# B&R Automation Studio project Praktyki_12_08
Automation Studio 4.12.5.95 SP; technology packages: mappCockpit 5.24.3, mappMotion 5.26.1, mappView 5.24.2

## Configuration Config1

CPU X20CP0484-1, AutomationRuntime K4.93, Build 4.1.2, Safety 0.0, Vc V4.72.6

### Task classes (Cpu.sw)
```
Cyclic#1:
  TCPXYZ <- PickAndPlace.TCPXYZ.prg
  Program <- PickAndPlace.Program.prg [disabled]
  PrgMechs <- PickAndPlace.PrgMechs.prg [disabled]
  PrgPickCor <- PickAndPlace.PrgPickCore.prg
  PrgPick <- PickAndPlace.PrgPick.prg
  PrgPlace <- PickAndPlace.PrgPlace.prg
DataObjects: McAcpSys
NcDataObjects: McDriveLog
Binaries: udbdef, arsvcreg, FWRules, McAcpDrv, McMechSys, McAcpSim, TCData, arflatprv, arcoal, visionUnit, mvLoader, McProfGen, mCoWebSc, TCLang, iomap, Config_4, asfw, Config_9, Config_3, Role, Config_8, Config_6, Config_7, Config_5, Config_1, Config_2, arconfig, ashwac, ashwd, Hierarchy, sysconf, User, Settings, Config_11, Config_10, Settings_1, viApp, viComp, Config_12, Config_13, Config
Libraries: McBase, MpBase, MpRobotics, McAxGroup, McPathGen, McAxis, McProgInt, McAcpAx, MpAxis, UserLib, MpPick, McTrkPath, CoTrace, AsZip, FileIO, runtime, Library, ViBase, AsARCfg, powerlnk, AsEPL, AsIO, sys_lib, DataObj, astime, McPureVAx, MpAlarmX, asmem, brsystem, asarprof, asarlog, asieccon, arssl
```

### Task classes (Cpu.sw)
```
Cyclic#4:
  PrgMechs <- PickAndPlace.PrgMechs.prg
  PrgPick <- PickAndPlace.PrgPick.prg
  PrgPlace <- PickAndPlace.PrgPlace.prg
  PrgPickCor <- PickAndPlace.PrgPickCore.prg
DataObjects: McAcpSys
NcDataObjects: McDriveLog
Binaries: McAcpDrv, udbdef, McAcpSim, mvLoader, arflatprv, McMechSys, TCData, mCoWebSc, FWRules, arcoal, arsvcreg, Settings, iomap, TraceConfi, ashwac, asfw, sysconf, arconfig, Config_6, Config_8, Hierarchy, ashwd, Role, Config_7, User, Config_9, Config_3, Config_1, Config_4, Config_2, Config_5, Config_14, Config_12, Config_10, Config_13, Config_11
Libraries: McBase, MpBase, MpRobotics, McAxGroup, McPathGen, McAxis, McProgInt, McAcpAx, CoTrace, AsZip, FileIO, runtime, MpAxis, MpPick, McTrkPath, asarprof, asieccon, asarlog, asio, asmem, astime, dataobj, asepl, brsystem, arssl, sys_lib, powerlnk
```

### Hardware
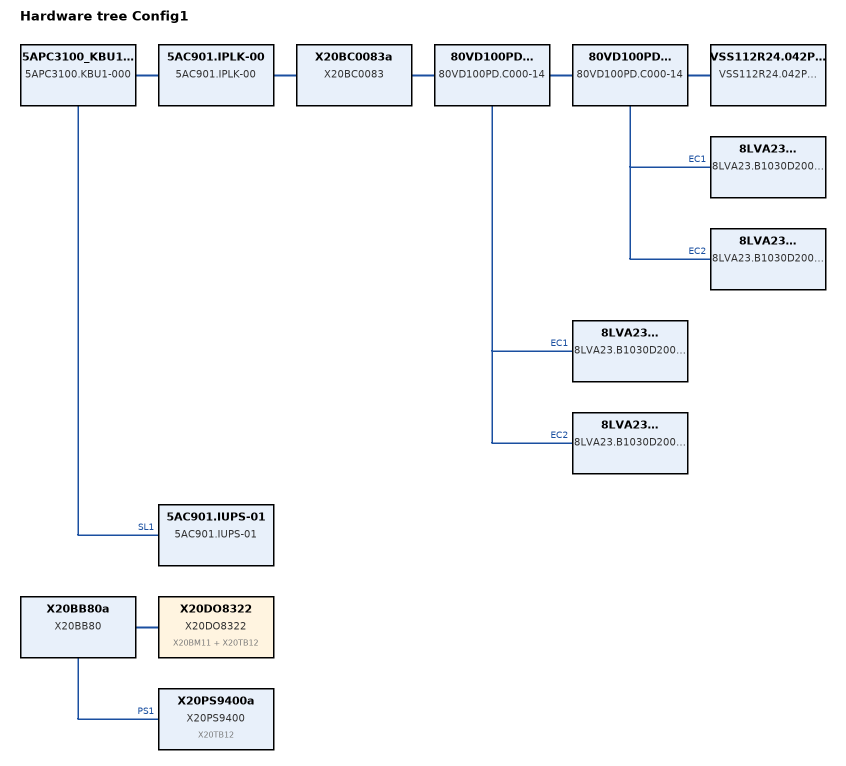
```
5AC901.IPLK-00 : 5AC901.IPLK-00 v1.8.0.1  [SL -> 5APC3100_KBU1_000.SL2]
  Connector IF1:
    MtuSize = 1500
    Channel1
    ChannelID1 = McAcpBroadcast
    ChannelType1 = OCTET[96]
    InternetAddress = 12.10.10.240
    SubnetMask = 255.255.255.0
5AC901.IUPS-01 : 5AC901.IUPS-01 v1.3.1.0  [SL -> 5APC3100_KBU1_000.SL1]
5APC3100_KBU1_000 : 5APC3100.KBU1-000 v2.2.1.0
  Connector IF3:
    AssignedOperatingSystem = ARemb
    ActivateDevice = 1
    Mode = Manual
    InternetAddress = 10.0.0.150
    SubnetMask = 255.255.255.0
    ActivateSnmp = 2
  Connector IF4:
    AssignedOperatingSystem = ARemb
    ActivateDevice = 1
    Mode = Manual
    InternetAddress = 192.168.0.20
    SubnetMask = 255.255.255.0
    ActivateSnmp = 2
  Connector IF5:
    AssignedOperatingSystem = ARemb
  Connector IF6:
    AssignedOperatingSystem = ARemb
  Connector IF7:
    AssignedOperatingSystem = ARemb
  Connector IF8:
    AssignedOperatingSystem = ARemb
  ConfigurationID = prawdziwaDelta_Config1
  Simulation = 1
  TimerDeviceType = EPLX2X
  TimerDevice = 5AC901.IPLK-00.IF1
  TaskClassIdleTime = 2000
  Cyclic1Tolerance = 0
  FileDevice1
  FileDeviceName1 = CNC_PrgDir
  FileDevicePath1 = USER_PATH
  FtpUser1
  FtpUsername1 = admin
  FtpUserPassword1 = q3LIg5ZPX9qKnYfEoKnLCuwwHRw0InMkB5MY3lkoy6s=
  FtpUserSalt1 = imXNidk5
  FTPAccessRight1 = 0
  ActivateOpcUa = 1
  OpcUaInformationModels_PV_Version = 1
80VD100PD.C000-14 : 80VD100PD.C000-14 v2.5.0.0  [PLK1 -> X20BC0083a.PLK2 (NodeNumber=1) [Cable Type=PowerlinkCable, Length=10, Version=1.0.0.3]; PLK2 -> 80VD100PD.C000-14a.PLK1 (NodeNumber=1) [Cable Type=PowerlinkCable, Length=10, Version=1.0.0.3]; EC1 -> 8LVA23.B1030D200-0.EC; EC2 -> 8LVA23.B1030D200-0a.EC; MT2 -> 8LVA23.B1030D200-0a.MT]
  DriveConfiguration/Module:
    McAcoposTypeID = AcoposMicroDConfig
    ActivateACOPOSSimulationOnPLC = 0
  DriveConfiguration/Channel[1]/RealAxis:
    AxisReference = gAxisQ1
    MechanicalElementsIsInvisible = 0
  DriveConfiguration/Channel[1]/RealAxis/MechanicalElements/Gearbox:
    InputIsReadOnly = 0
    Input = 25
    OutputIsReadOnly = 0
    Output = 1
  DriveConfiguration/Channel[1]/RealAxis/MechanicalElements/RotaryToLinearTransformation:
    ReferenceDistanceIsReadOnly = 0
    ReferenceDistance = 1
  DriveConfiguration/Channel[1]/RealAxis/Controller:
    ModeIsReadOnly = 0
    Mode = PositionController
  DriveConfiguration/Channel[1]/RealAxis/Controller/Mode/Position:
    ProportionalGain = 402
    IntegrationTime = 0.0
    PredictionTime = 0.0004
    TotalDelayTime = 0.0004
  DriveConfiguration/Channel[1]/RealAxis/Controller/Mode/Speed:
    ProportionalGainIsReadOnly = 0
    ProportionalGain = 1.7
    IntegrationTimeIsReadOnly = 0
    IntegrationTime = 0.0
    FilterTimeIsReadOnly = 0
    FilterTime = 0.0
  DriveConfiguration/Channel[1]/RealAxis/Controller/Mode/LoopFilters:
    LoopFilterXIsReadOnly = 0
    LoopFilter1 = NotUsed
    LoopFilter2 = NotUsed
    LoopFilter3 = NotUsed
  DriveConfiguration/Channel[1]/RealAxis/Homing:
    ModeIsReadOnly = 0
    Mode = Absolute
  DriveConfiguration/Channel[1]/RealAxis/Homing/Mode:
    Position = 0
  DriveConfiguration/Channel[1]/RealAxis/Homing:
    RestorePositionVariable = 
  DriveConfiguration/Channel[1]/RealAxis/StopReaction:
    QuickstopIsReadOnly = 0
    Quickstop = DecelerationLimit
    DriveErrorIsReadOnly = 0
    DriveError = DecelerationLimit
  DriveConfiguration/Channel[1]/RealAxis/MovementErrorLimits:
    PositionError = 1.0
    VelocityErrorMonitoring = Automatic1
  DriveConfiguration/Channel[1]/RealAxis:
    JerkFilterIsReadOnly = 0
    JerkFilter = NotUsed
    ZeroVibrationFilter = NotUsed
  DriveConfiguration/Channel[1]/RealAxis/DigitalInputs/HomingSwitch:
    SourceIsReadOnly = 0
    Source = NotUsed
    Level = High
  DriveConfiguration/Channel[1]/RealAxis/DigitalInputs/PositiveLimitSwitch:
    SourceIsReadOnly = 0
    Source = NotUsed
    Level = High
  DriveConfiguration/Channel[1]/RealAxis/DigitalInputs/NegativeLimitSwitch:
    SourceIsReadOnly = 0
    Source = NotUsed
    Level = High
  DriveConfiguration/Channel[1]/RealAxis/DigitalInputs/Trigger1:
    Source = X2Trigger1
    Level = High
  DriveConfiguration/Channel[1]/RealAxis/DigitalInputs/Trigger2:
    Source = X2Trigger2
    Level = High
  DriveConfiguration/Channel[1]/RealAxis/DigitalInputs/Quickstop:
    Input = Trigger2
  DriveConfiguration/Channel[1]/RealAxis/Simulation:
    SimulationModeOnPLC = SetValueGeneration
    SimulationModeOnACOPOS = NotUsed
  DriveConfiguration/Channel[1]:
    ExternalEncoderAxis = NotUsed
  DriveConfiguration/Channel[2]/RealAxis:
    AxisReference = gAxisQ2
    MechanicalElementsIsInvisible = 0
  DriveConfiguration/Channel[2]/RealAxis/MechanicalElements/Gearbox:
    InputIsReadOnly = 0
    Input = 25
    OutputIsReadOnly = 0
    Output = 1
  DriveConfiguration/Channel[2]/RealAxis/MechanicalElements/RotaryToLinearTransformation:
    ReferenceDistanceIsReadOnly = 0
    ReferenceDistance = 1
  DriveConfiguration/Channel[2]/RealAxis/Controller:
    ModeIsReadOnly = 0
    Mode = PositionController
  DriveConfiguration/Channel[2]/RealAxis/Controller/Mode/Position:
    ProportionalGain = 393
    IntegrationTime = 0.0
    PredictionTime = 0.0004
    TotalDelayTime = 0.0004
  DriveConfiguration/Channel[2]/RealAxis/Controller/Mode/Speed:
    ProportionalGainIsReadOnly = 0
    ProportionalGain = 1.65
    IntegrationTimeIsReadOnly = 0
    IntegrationTime = 0.0
    FilterTimeIsReadOnly = 0
    FilterTime = 0.0
  DriveConfiguration/Channel[2]/RealAxis/Controller/Mode/LoopFilters:
    LoopFilterXIsReadOnly = 0
    LoopFilter1 = NotUsed
    LoopFilter2 = NotUsed
    LoopFilter3 = NotUsed
  DriveConfiguration/Channel[2]/RealAxis/Homing:
    ModeIsReadOnly = 0
    Mode = Absolute
  DriveConfiguration/Channel[2]/RealAxis/Homing/Mode:
    Position = 0
  DriveConfiguration/Channel[2]/RealAxis/Homing:
    RestorePositionVariable = 
  DriveConfiguration/Channel[2]/RealAxis/StopReaction:
    QuickstopIsReadOnly = 0
    Quickstop = DecelerationLimit
    DriveErrorIsReadOnly = 0
    DriveError = DecelerationLimit
  DriveConfiguration/Channel[2]/RealAxis/MovementErrorLimits:
    PositionError = 1.0
    VelocityErrorMonitoring = Automatic1
  DriveConfiguration/Channel[2]/RealAxis:
    JerkFilterIsReadOnly = 0
    JerkFilter = NotUsed
    ZeroVibrationFilter = NotUsed
  DriveConfiguration/Channel[2]/RealAxis/DigitalInputs/HomingSwitch:
    SourceIsReadOnly = 0
    Source = NotUsed
    Level = High
  DriveConfiguration/Channel[2]/RealAxis/DigitalInputs/PositiveLimitSwitch:
    SourceIsReadOnly = 0
    Source = NotUsed
    Level = High
  DriveConfiguration/Channel[2]/RealAxis/DigitalInputs/NegativeLimitSwitch:
    SourceIsReadOnly = 0
    Source = NotUsed
    Level = High
  DriveConfiguration/Channel[2]/RealAxis/DigitalInputs/Trigger1:
    Source = X2Trigger1
    Level = High
  DriveConfiguration/Channel[2]/RealAxis/DigitalInputs/Trigger2:
    Source = X2Trigger2
    Level = High
  DriveConfiguration/Channel[2]/RealAxis/DigitalInputs/Quickstop:
    Input = Trigger2
  DriveConfiguration/Channel[2]/RealAxis/Simulation:
    SimulationModeOnPLC = SetValueGeneration
    SimulationModeOnACOPOS = NotUsed
  DriveConfiguration/Channel[2]:
    ExternalEncoderAxis = NotUsed
80VD100PD.C000-14a : 80VD100PD.C000-14 v2.5.0.0  [PLK1 -> 80VD100PD.C000-14.PLK2 (NodeNumber=2) [Cable Type=PowerlinkCable, Length=10, Version=1.0.0.3]; PLK2 -> VSS112R24.042P-000.PLK1 (NodeNumber=2) [Cable Type=PowerlinkCable, Length=10, Version=1.0.0.3]; EC1 -> 8LVA23.B1030D200-0b.EC; EC2 -> 8LVA23.B1030D200-0c.EC; MT2 -> 8LVA23.B1030D200-0c.MT]
  DriveConfiguration/Module:
    McAcoposTypeID = AcoposMicroDConfig
    ActivateACOPOSSimulationOnPLC = 0
  DriveConfiguration/Channel[1]/RealAxis:
    AxisReference = gAxisQ3
    MechanicalElementsIsInvisible = 0
  DriveConfiguration/Channel[1]/RealAxis/MechanicalElements/Gearbox:
    InputIsReadOnly = 0
    Input = 25
    OutputIsReadOnly = 0
    Output = 1
  DriveConfiguration/Channel[1]/RealAxis/MechanicalElements/RotaryToLinearTransformation:
    ReferenceDistanceIsReadOnly = 0
    ReferenceDistance = 1
  DriveConfiguration/Channel[1]/RealAxis/Controller:
    ModeIsReadOnly = 0
    Mode = PositionController
  DriveConfiguration/Channel[1]/RealAxis/Controller/Mode/Position:
    ProportionalGain = 400
    IntegrationTime = 0.0
    PredictionTime = 0.0004
    TotalDelayTime = 0.0004
  DriveConfiguration/Channel[1]/RealAxis/Controller/Mode/Speed:
    ProportionalGainIsReadOnly = 0
    ProportionalGain = 1.7
    IntegrationTimeIsReadOnly = 0
    IntegrationTime = 0.0
    FilterTimeIsReadOnly = 0
    FilterTime = 0.0
  DriveConfiguration/Channel[1]/RealAxis/Controller/Mode/LoopFilters:
    LoopFilterXIsReadOnly = 0
    LoopFilter1 = NotUsed
    LoopFilter2 = NotUsed
    LoopFilter3 = NotUsed
  DriveConfiguration/Channel[1]/RealAxis/Homing:
    ModeIsReadOnly = 0
    Mode = Absolute
  DriveConfiguration/Channel[1]/RealAxis/Homing/Mode:
    Position = 0
  DriveConfiguration/Channel[1]/RealAxis/Homing:
    RestorePositionVariable = 
  DriveConfiguration/Channel[1]/RealAxis/StopReaction:
    QuickstopIsReadOnly = 0
    Quickstop = DecelerationLimit
    DriveErrorIsReadOnly = 0
    DriveError = DecelerationLimit
  DriveConfiguration/Channel[1]/RealAxis/MovementErrorLimits:
    PositionError = 1.0
    VelocityErrorMonitoring = Automatic1
  DriveConfiguration/Channel[1]/RealAxis:
    JerkFilterIsReadOnly = 0
    JerkFilter = NotUsed
    ZeroVibrationFilter = NotUsed
  DriveConfiguration/Channel[1]/RealAxis/DigitalInputs/HomingSwitch:
    SourceIsReadOnly = 0
    Source = NotUsed
    Level = High
  DriveConfiguration/Channel[1]/RealAxis/DigitalInputs/PositiveLimitSwitch:
    SourceIsReadOnly = 0
    Source = NotUsed
    Level = High
  DriveConfiguration/Channel[1]/RealAxis/DigitalInputs/NegativeLimitSwitch:
    SourceIsReadOnly = 0
    Source = NotUsed
    Level = High
  DriveConfiguration/Channel[1]/RealAxis/DigitalInputs/Trigger1:
    Source = X2Trigger1
    Level = High
  DriveConfiguration/Channel[1]/RealAxis/DigitalInputs/Trigger2:
    Source = X2Trigger2
    Level = High
  DriveConfiguration/Channel[1]/RealAxis/DigitalInputs/Quickstop:
    Input = Trigger2
  DriveConfiguration/Channel[1]/RealAxis/Simulation:
    SimulationModeOnPLC = SetValueGeneration
    SimulationModeOnACOPOS = NotUsed
  DriveConfiguration/Channel[1]:
    ExternalEncoderAxis = NotUsed
  DriveConfiguration/Channel[2]/RealAxis:
    AxisReference = gAxis_1
    MechanicalElementsIsInvisible = 0
  DriveConfiguration/Channel[2]/RealAxis/MechanicalElements/Gearbox:
    InputIsReadOnly = 0
    Input = 1
    OutputIsReadOnly = 0
    Output = 1
  DriveConfiguration/Channel[2]/RealAxis/MechanicalElements/RotaryToLinearTransformation:
    ReferenceDistanceIsReadOnly = 0
    ReferenceDistance = 1
  DriveConfiguration/Channel[2]/RealAxis/Controller:
    ModeIsReadOnly = 0
    Mode = PositionController
  DriveConfiguration/Channel[2]/RealAxis/Controller/Mode/Position:
    ProportionalGain = 50.0
    IntegrationTime = 0.0
    PredictionTime = 0.0004
    TotalDelayTime = 0.0004
  DriveConfiguration/Channel[2]/RealAxis/Controller/Mode/Speed:
    ProportionalGainIsReadOnly = 0
    ProportionalGain = 2.0
    IntegrationTimeIsReadOnly = 0
    IntegrationTime = 0.0
    FilterTimeIsReadOnly = 0
    FilterTime = 0.0
  DriveConfiguration/Channel[2]/RealAxis/Controller/Mode/LoopFilters:
    LoopFilterXIsReadOnly = 0
    LoopFilter1 = NotUsed
    LoopFilter2 = NotUsed
    LoopFilter3 = NotUsed
  DriveConfiguration/Channel[2]/RealAxis/Homing:
    ModeIsReadOnly = 0
    Mode = Direct
  DriveConfiguration/Channel[2]/RealAxis/Homing/Mode:
    Position = 0.0
    ReferencePulse = NotUsed
  DriveConfiguration/Channel[2]/RealAxis/Homing:
    RestorePositionVariable = 
  DriveConfiguration/Channel[2]/RealAxis/StopReaction:
    QuickstopIsReadOnly = 0
    Quickstop = DecelerationLimit
    DriveErrorIsReadOnly = 0
    DriveError = DecelerationLimit
  DriveConfiguration/Channel[2]/RealAxis/MovementErrorLimits:
    PositionError = 1.0
    VelocityErrorMonitoring = Automatic1
  DriveConfiguration/Channel[2]/RealAxis:
    JerkFilterIsReadOnly = 0
    JerkFilter = NotUsed
    ZeroVibrationFilter = NotUsed
  DriveConfiguration/Channel[2]/RealAxis/DigitalInputs/HomingSwitch:
    SourceIsReadOnly = 0
    Source = NotUsed
    Level = High
  DriveConfiguration/Channel[2]/RealAxis/DigitalInputs/PositiveLimitSwitch:
    SourceIsReadOnly = 0
    Source = NotUsed
    Level = High
  DriveConfiguration/Channel[2]/RealAxis/DigitalInputs/NegativeLimitSwitch:
    SourceIsReadOnly = 0
    Source = NotUsed
    Level = High
  DriveConfiguration/Channel[2]/RealAxis/DigitalInputs/Trigger1:
    Source = X2Trigger1
    Level = High
  DriveConfiguration/Channel[2]/RealAxis/DigitalInputs/Trigger2:
    Source = X2Trigger2
    Level = High
  DriveConfiguration/Channel[2]/RealAxis/DigitalInputs/Quickstop:
    Input = Trigger2
  DriveConfiguration/Channel[2]/RealAxis/Simulation:
    SimulationModeOnPLC = SetValueGeneration
    SimulationModeOnACOPOS = NotUsed
  DriveConfiguration/Channel[2]:
    ExternalEncoderAxis = NotUsed
8LVA23.B1030D200-0 : 8LVA23.B1030D200-0 v2.2.0.3  [EC -> 80VD100PD.C000-14.EC1; MT -> 80VD100PD.C000-14.MT1]
  M1/MotorParameters:
    MOTOR_AMB_TEMP_RATED = 40
8LVA23.B1030D200-0a : 8LVA23.B1030D200-0 v2.2.0.3  [EC -> 80VD100PD.C000-14.EC2; MT -> 80VD100PD.C000-14.MT2]
  M1/MotorParameters:
    MOTOR_AMB_TEMP_RATED = 40
8LVA23.B1030D200-0b : 8LVA23.B1030D200-0 v2.2.0.3  [EC -> 80VD100PD.C000-14a.EC1; MT -> 80VD100PD.C000-14a.MT1]
  M1/MotorParameters:
    MOTOR_AMB_TEMP_RATED = 40
8LVA23.B1030D200-0c : 8LVA23.B1030D200-0 v2.2.0.3  [EC -> 80VD100PD.C000-14a.EC2; MT -> 80VD100PD.C000-14a.MT2]
  M1/MotorParameters:
    MOTOR_AMB_TEMP_RATED = 40
VSS112R24.042P-000 : VSS112R24.042P-000 v1.9.0.730  [PLK1 -> 80VD100PD.C000-14a.PLK2 (NodeNumber=4) [Cable Type=PowerlinkCable, Length=10, Version=1.0.0.3]]
  Supervision = off
  VisionConfig = gCamera
X20BB80a : X20BB80 v1.1.0.0
X20BC0083a : X20BC0083 v2.14.0.0  [PLK1 -> 5AC901.IPLK-00.IF1 (NodeNumber=3) [Cable Type=PowerlinkCable, Length=10, Version=1.0.0.3]; PLK2 -> 80VD100PD.C000-14.PLK1 (NodeNumber=3) [Cable Type=PowerlinkCable, Length=10, Version=1.0.0.3]; SL -> X20BB80a.SL1]
  Supervision = off
X20BM11a : X20BM11 v1.1.0.0  [X2X1 -> X20BB80a.IF1]
X20DO8322 : X20DO8322 v1.5.0.0  [SS1 -> X20TB12b.SS; SL -> X20BM11a.SL1]
X20PS9400a : X20PS9400 v1.8.0.0  [SS1 -> X20TB12a.SS; PS -> X20BB80a.PS1]
  Supervision = off
X20TB12a : X20TB12 v1.0.0.0
X20TB12b : X20TB12 v1.0.0.0
```

### IoMap.iom - 5APC3100_KBU1_000/IoMap.iom
```iecst
VAR_CONFIG
	::Gripper AT %QX."X20DO8322".DigitalOutput08;
END_VAR
```

### Config_1.axesgroup - 5APC3100_KBU1_000/mappMotion/4AxesDeltaA/Config_1.axesgroup
```
Element g4AxDeltaA (Type=axesgroup)
  Type = PathGenAxesGroup
    ProcessingTaskClass = 255
    License = 1
    PhysicalAxes:
      JointAxes:
        JointAxisAxisRefIsReadOnly = 0
        JointAxis[1]:
          Name = Q1
          AxisRef = gAxisQ1
        JointAxis[2]:
          Name = Q2
          AxisRef = gAxisQ2
        JointAxis[3]:
          Name = Q3
          AxisRef = gAxisQ3
        JointAxis[4]:
          Name = Q4
          AxisRef = gAxisQ4
    MechanicalSystem:
      MechSysRefIsReadOnly = 0
      MechSysRef = MechSys_4AxDeltaA
    BasicSettings:
      ModalDataBehaviour = ResetToDefault
      GeometryPlanning:
        TCPResolutionIsReadOnly = 0
        TCPResolution:
          LengthResolution = 0.001
          AngleResolution = 0.001
        Rounding:
          PathDistance = 0.0
          SymmetricRounding = Yes
          LastSegment = Half
          AvoidZeroCurvature = No
        RoundingMode = Standard
        MaxCornerDeviation = 0.0
        MaxTangentialTransitionDeviation = 0.0
        MaxRadiusDeviation = 0.001
        WorkingPlane = XY
      TrajectoryPlanningIsReadOnly = 0
      TrajectoryPlanning = Basic
        LimitCheckResolutionIsReadOnly = 0
        LimitCheckResolution = Automatic
        BufferTime = Automatic
        BarrierParametrization = JointCoordinates
        TorqueLimitConsideration = Exact
      Miscellaneous:
        NonMovementsLimit = NotUsed
        TimeStretchOverride:
          JerkSuppression = NotUsed
    StopReaction:
      AxisError:
        AxisReactionIsReadOnly = 0
    AxesGroupFeatures:
      FeatureRef[1] = Feature_Programs
      FeatureRef[2] = Feature_Jogging
      FeatureRef[3] = Feature_FrameHierarchy
      FeatureRef[4] = Feature_Tracking
      FeatureRef[5] = Feature_PathDefinition
  Alarms = MpAlarmX
```

### Config_2.axis - 5APC3100_KBU1_000/mappMotion/4AxesDeltaA/Config_2.axis
```
Element gAxisQ1 (Type=axis)
  BaseTypeIsReadOnly = 0
  BaseType = RotaryBounded
    MeasurementUnitIsReadOnly = 0
    MeasurementUnit = 17476
    MeasurementResolutionIsReadOnly = 0
    MeasurementResolution = 0.01
    CountDirectionIsReadOnly = 0
    CountDirection = Standard
  MovementLimitsIsReadOnly = 0
  MovementLimits = InternalForPathControlledAxis
    Position:
      LowerLimitMin = -1.79769313486231E308
      UpperLimitMax = 1.79769313486231E308
      LowerLimit = -90
      UpperLimit = 110
    VelocityIsReadOnly = 0
    Velocity:
      VelocityMax = 3.4E38
      Velocity = 50000
    AccelerationIsReadOnly = 0
    Acceleration:
      AccelerationMax = 3.4E38
      Acceleration = 500000
    DecelerationIsReadOnly = 0
    Deceleration:
      DecelerationMax = 3.4E38
      Deceleration = 500000
    JerkIsReadOnly = 0
    Jerk = Basic
      JerkMax = 3.4E38
      Jerk = 500000
    TorqueIsInvisible = 0
    TorqueIsReadOnly = 0
  Alarms = None
Element gAxisQ2 (Type=axis)
  BaseTypeIsReadOnly = 0
  BaseType = RotaryBounded
    MeasurementUnitIsReadOnly = 0
    MeasurementUnit = 17476
    MeasurementResolutionIsReadOnly = 0
    MeasurementResolution = 0.01
    CountDirectionIsReadOnly = 0
    CountDirection = Inverse
  MovementLimitsIsReadOnly = 0
  MovementLimits = InternalForPathControlledAxis
    Position:
      LowerLimitMin = -1.79769313486231E308
      UpperLimitMax = 1.79769313486231E308
      LowerLimit = -90
      UpperLimit = 110
    VelocityIsReadOnly = 0
    Velocity:
      VelocityMax = 3.4E38
      Velocity = 50000
    AccelerationIsReadOnly = 0
    Acceleration:
      AccelerationMax = 3.4E38
      Acceleration = 500000
    DecelerationIsReadOnly = 0
    Deceleration:
      DecelerationMax = 3.4E38
      Deceleration = 500000
    JerkIsReadOnly = 0
    Jerk = Basic
      JerkMax = 3.4E38
      Jerk = 500000
    TorqueIsInvisible = 0
    TorqueIsReadOnly = 0
  Alarms = None
Element gAxisQ3 (Type=axis)
  BaseTypeIsReadOnly = 0
  BaseType = RotaryBounded
    MeasurementUnitIsReadOnly = 0
    MeasurementUnit = 17476
    MeasurementResolutionIsReadOnly = 0
    MeasurementResolution = 0.01
    CountDirectionIsReadOnly = 0
    CountDirection = Inverse
  MovementLimitsIsReadOnly = 0
  MovementLimits = InternalForPathControlledAxis
    Position:
      LowerLimitMin = -1.79769313486231E308
      UpperLimitMax = 1.79769313486231E308
      LowerLimit = -90
      UpperLimit = 110
    VelocityIsReadOnly = 0
    Velocity:
      VelocityMax = 3.4E38
      Velocity = 50000
    AccelerationIsReadOnly = 0
    Acceleration:
      AccelerationMax = 3.4E38
      Acceleration = 500000
    DecelerationIsReadOnly = 0
    Deceleration:
      DecelerationMax = 3.4E38
      Deceleration = 500000
    JerkIsReadOnly = 0
    Jerk = Basic
      JerkMax = 3.4E38
      Jerk = 500000
    TorqueIsInvisible = 0
    TorqueIsReadOnly = 0
  Alarms = None
Element gAxisQ4 (Type=axis)
  BaseTypeIsReadOnly = 0
  BaseType = Rotary
    MeasurementUnitIsReadOnly = 0
    MeasurementUnit = 17476
    MeasurementResolutionIsReadOnly = 0
    MeasurementResolution = 0.01
    CountDirectionIsReadOnly = 0
    CountDirection = Standard
  MovementLimitsIsReadOnly = 0
  MovementLimits = InternalForPathControlledAxis
    Position:
      LowerLimitMin = -1.79769313486231E308
      UpperLimitMax = 1.79769313486231E308
      LowerLimit = -1000.0
      UpperLimit = 1000.0
    VelocityIsReadOnly = 0
    Velocity:
      VelocityMax = 3.4E38
      Velocity = 5000
    AccelerationIsReadOnly = 0
    Acceleration:
      AccelerationMax = 3.4E38
      Acceleration = 50000
    DecelerationIsReadOnly = 0
    Deceleration:
      DecelerationMax = 3.4E38
      Deceleration = 50000
    JerkIsReadOnly = 0
    Jerk = Basic
      JerkMax = 3.4E38
      Jerk = 500000
    TorqueIsInvisible = 0
    TorqueIsReadOnly = 0
  Alarms = MpAlarmX
```

### Config_3.mechanicalsystem - 5APC3100_KBU1_000/mappMotion/4AxesDeltaA/Config_3.mechanicalsystem
```
Element MechSys_4AxDeltaA (Type=mechanicalsystem)
  TypeIsReadOnly = 0
  Type = Delta
    SubtypeIsReadOnly = 0
    Subtype = 4AxesDeltaA
      SceneViewerObject = Generic
      DescriptionIsReadOnly = 0
      Description = Standard
        Dimensions:
          BasePlatform:
            CenterIsReadOnly = 0
            Center:
              X = 0.0
              Y = 0.0
              Z = 0.0
            ArmLinkPointIsReadOnly = 0
            Arm1LinkPoint:
              Angle = 0.0
              Radius = 250.0
              Z = 0.0
            Arm2LinkPoint:
              Angle = 90
              Radius = 250.0
              Z = 0.0
            Arm3LinkPoint:
              Angle = 180
              Radius = 250.0
              Z = 0.0
          Arms:
            ArmIsReadOnly = 0
            Arm1:
              UpperArmLength = 600.0
              LowerArmLength = 900.0
            Arm2:
              UpperArmLength = 600.0
              LowerArmLength = 900.0
            Arm3:
              UpperArmLength = 600.0
              LowerArmLength = 900.0
            LowerArmPairDistance = 0.0
          EndEffectorPlatform:
            ArmLinkPointIsReadOnly = 0
            Arm1LinkPoint:
              Radius = 50.0
              Z = 0.0
            Arm2LinkPoint:
              Radius = 50.0
              Z = 0.0
            Arm3LinkPoint:
              Radius = 50.0
              Z = 0.0
            TranslationToFlangeIsReadOnly = 0
            TranslationToFlange:
              X = 0.0
              Y = 0.0
              Z = -150
        Offsets:
          JointAxisIsReadOnly = 0
          JointAxis[1] = 0.0
          JointAxis[2] = 0.0
          JointAxis[3] = 0.0
          JointAxis[4] = 0.0
        CountDirections:
          JointAxisIsReadOnly = 0
          JointAxis[1] = Standard
          JointAxis[2] = Standard
          JointAxis[3] = Standard
          JointAxis[4] = Standard
      CoordinatesNames = Default
        XCoordinateName = X
        YCoordinateName = Y
        ZCoordinateName = Z
        CCoordinateName = C
      TcpOrientation:
        Frames = Used
      WireFrameModelIsReadOnly = 0
      WireFrameModel = Standard
        UpperArm1IsReadOnly = 0
        UpperArm1 = ConnectionLine
          DistanceMin = -1.79769313486231E308
          DistanceMax = 1.79769313486231E308
          Distance = 0.0
        LowerArm1IsReadOnly = 0
        LowerArm1 = ConnectionLine
          DistanceMin = -1.79769313486231E308
          DistanceMax = 1.79769313486231E308
          Distance = 0.0
        UpperArm2IsReadOnly = 0
        UpperArm2 = ConnectionLine
          DistanceMin = -1.79769313486231E308
          DistanceMax = 1.79769313486231E308
          Distance = 0.0
        LowerArm2IsReadOnly = 0
        LowerArm2 = ConnectionLine
          DistanceMin = -1.79769313486231E308
          DistanceMax = 1.79769313486231E308
          Distance = 0.0
        UpperArm3IsReadOnly = 0
        UpperArm3 = ConnectionLine
          DistanceMin = -1.79769313486231E308
          DistanceMax = 1.79769313486231E308
          Distance = 0.0
        LowerArm3IsReadOnly = 0
        LowerArm3 = ConnectionLine
          DistanceMin = -1.79769313486231E308
          DistanceMax = 1.79769313486231E308
          Distance = 0.0
        EndEffectorPlatformToFlangeIsReadOnly = 0
        EndEffectorPlatformToFlange = ConnectionLine
          DistanceMin = -1.79769313486231E308
          DistanceMax = 1.79769313486231E308
          Distance = 0.0
        FlangeToTcp = ConnectionLine
          DistanceMin = -1.79769313486231E308
          DistanceMax = 1.79769313486231E308
          Distance = 0.0
      DynamicModelIsReadOnly = 0
      DynamicModel = DynParTable
        TableRef
      InternalDynamicModelIsReadOnly = 0
      InternalDynamicModel = NotUsed
      DynamicLimits = DynParTables
        GearboxLimitsTableRef
        CrossSectionLimitsTableRef
      InternalDynamicLimits = NotUsed
      LoadDependentJerkLimitsIsReadOnly = 0
      LoadDependentJerkLimits = NotUsed
      CouplingsIsInvisible = 0
      JointAxesPositionLimits:
        JointAxisIsReadOnly = 0
        JointAxis[1] = UseAxisLimits
        JointAxis[2] = UseAxisLimits
        JointAxis[3] = UseAxisLimits
        JointAxis[4] = UseAxisLimits
      WorkingRangeIsReadOnly = 0
      WorkingRange = Standard
        BaseToTopIsReadOnly = 0
        BaseToTop = 400
        TopHeightIsReadOnly = 0
        TopHeight = 100
        MiddleHeightIsReadOnly = 0
        MiddleHeight = 400
        BottomHeightIsReadOnly = 0
        BottomHeight = 600
        TopRadiusIsReadOnly = 0
        TopRadius = 800
        MiddleRadiusIsReadOnly = 0
        MiddleRadius = 900
        BottomRadiusIsReadOnly = 0
        BottomRadius = 200
```

### Config_5.axis - 5APC3100_KBU1_000/mappMotion/4AxesDeltaA/Config_5.axis
```
Element gAxis_1 (Type=axis)
  BaseTypeIsReadOnly = 0
  BaseType = LinearPeriodic
    MeasurementUnit = 5066068
    MeasurementResolutionIsReadOnly = 0
    MeasurementResolution = 0.01
    CountDirectionIsReadOnly = 0
    CountDirection = Inverse
    PeriodSettings:
      Period = 2000
  MovementLimitsIsReadOnly = 0
  MovementLimits = Internal
    Position:
      LowerLimitMin = -1.79769313486231E308
      UpperLimitMax = 1.79769313486231E308
      LowerLimit = -1000.0
      UpperLimit = 1000.0
    VelocityIsReadOnly = 0
    Velocity:
      VelocityMax = 3.4E38
      Velocity = 5000
    AccelerationIsReadOnly = 0
    Acceleration:
      AccelerationMax = 3.4E38
      Acceleration = 50000
    DecelerationIsReadOnly = 0
    Deceleration:
      DecelerationMax = 3.4E38
      Deceleration = 50000
  Alarms = MpAlarmX
    mapp.AlarmX.Core.Configuration:
      [0]:
        Message = System problem - ConveyorPick
      [1]:
        Message = Initialization problem - ConveyorPick
      [2]:
        Message = Parameter problem - ConveyorPick
      [3]:
        Message = Operation problem - ConveyorPick
      [4]:
        Message = Data access problem - ConveyorPick
      [5]:
        Message = Syntax error - ConveyorPick
      [9]:
        Message = Network problem - ConveyorPick
      [10]:
        Message = Encoder problem - ConveyorPick
      [11]:
        Message = Drive problem - ConveyorPick
      [12]:
        Message = IO problem - ConveyorPick
      [13]:
        Message = Supply problem - ConveyorPick
      [14]:
        Message = Motor problem - ConveyorPick
      [15]:
        Message = Holding brake problem - ConveyorPick
      [19]:
        Message = Movement error limit reached - ConveyorPick
      [20]:
        Message = HW or SW movement limits reached - ConveyorPick
      [21]:
        Message = Enable input low - ConveyorPick
Element gAxis_2 (Type=axis)
  BaseTypeIsReadOnly = 0
  BaseType = LinearPeriodic
    MeasurementUnit = 5066068
    MeasurementResolutionIsReadOnly = 0
    MeasurementResolution = 0.01
    CountDirectionIsReadOnly = 0
    CountDirection = Standard
    PeriodSettings:
      Period = 2000
  MovementLimitsIsReadOnly = 0
  MovementLimits = Internal
    Position:
      LowerLimitMin = -1.79769313486231E308
      UpperLimitMax = 1.79769313486231E308
      LowerLimit = -1000.0
      UpperLimit = 1000.0
    VelocityIsReadOnly = 0
    Velocity:
      VelocityMax = 3.4E38
      Velocity = 1
    AccelerationIsReadOnly = 0
    Acceleration:
      AccelerationMax = 3.4E38
      Acceleration = 1
    DecelerationIsReadOnly = 0
    Deceleration:
      DecelerationMax = 3.4E38
      Deceleration = 1
  Alarms = MpAlarmX
    mapp.AlarmX.Core.Configuration:
      [0]:
        Message = System problem - PlaceHolder
      [1]:
        Message = Initialization problem - PlaceHolder
      [2]:
        Message = Parameter problem - PlaceHolder
      [3]:
        Message = Operation problem - PlaceHolder
      [4]:
        Message = Data access problem - PlaceHolder
      [5]:
        Message = Syntax error - PlaceHolder
      [9]:
        Message = Network problem - PlaceHolder
      [10]:
        Message = Encoder problem - PlaceHolder
      [11]:
        Message = Drive problem - PlaceHolder
      [12]:
        Message = IO problem - PlaceHolder
      [13]:
        Message = Supply problem - PlaceHolder
      [14]:
        Message = Motor problem - PlaceHolder
      [15]:
        Message = Holding brake problem - PlaceHolder
      [19]:
        Message = Movement error limit reached - PlaceHolder
      [20]:
        Message = HW or SW movement limits reached - PlaceHolder
      [21]:
        Message = Enable input low - PlaceHolder
Element gAxis_3 (Type=axis)
  BaseTypeIsReadOnly = 0
  BaseType = LinearBounded
    MeasurementUnit = 5066068
    MeasurementResolutionIsReadOnly = 0
    MeasurementResolution = 0.01
    CountDirectionIsReadOnly = 0
    CountDirection = Standard
  MovementLimitsIsReadOnly = 0
  MovementLimits = Internal
    Position:
      LowerLimitMin = -1.79769313486231E308
      UpperLimitMax = 1.79769313486231E308
      LowerLimit = -1000.0
      UpperLimit = 1000.0
    VelocityIsReadOnly = 0
    Velocity:
      VelocityMax = 3.4E38
      Velocity = 10.0
    AccelerationIsReadOnly = 0
    Acceleration:
      AccelerationMax = 3.4E38
      Acceleration = 50.0
    DecelerationIsReadOnly = 0
    Deceleration:
      DecelerationMax = 3.4E38
      Deceleration = 50.0
  Alarms = MpAlarmX
```

### Config_10.purevaxcfg - 5APC3100_KBU1_000/mappMotion/Config_10.purevaxcfg
```
Element PureVAxCfg_1 (Type=purevaxcfg)
  TypeID = PureVAxConfig
  PureVAxis:
    AxisReference = gAxisQ4
    Homing:
      Mode = Direct
        Position = 0.0
        ReferencePulse = NotUsed
      RestorePositionVariable
    JerkFilter = NotUsed
    ZeroVibrationFilter = NotUsed
```

### Config_11.purevaxcfg - 5APC3100_KBU1_000/mappMotion/Config_11.purevaxcfg
```
Element PureVAxCfg_2 (Type=purevaxcfg)
  TypeID = PureVAxConfig
  PureVAxis:
    AxisReference = gAxis_2
    Homing:
      Mode = Direct
        Position = 0.0
        ReferencePulse = NotUsed
      RestorePositionVariable
    JerkFilter = NotUsed
    ZeroVibrationFilter = NotUsed
```

### Config_5.axis - 5APC3100_KBU1_000/mappMotion/Config_5.axis
```
Element gAxis_1 (Type=axis)
  BaseTypeIsReadOnly = 0
  BaseType = LinearPeriodic
    MeasurementUnit = 5066068
    MeasurementResolutionIsReadOnly = 0
    MeasurementResolution = 0.01
    CountDirectionIsReadOnly = 0
    CountDirection = Inverse
    PeriodSettings:
      Period = 2000
  MovementLimitsIsReadOnly = 0
  MovementLimits = Internal
    Position:
      LowerLimitMin = -1.79769313486231E308
      UpperLimitMax = 1.79769313486231E308
      LowerLimit = -1000.0
      UpperLimit = 1000.0
    VelocityIsReadOnly = 0
    Velocity:
      VelocityMax = 3.4E38
      Velocity = 500
    AccelerationIsReadOnly = 0
    Acceleration:
      AccelerationMax = 3.4E38
      Acceleration = 5000
    DecelerationIsReadOnly = 0
    Deceleration:
      DecelerationMax = 3.4E38
      Deceleration = 50000
  Alarms = None
Element gAxis_2 (Type=axis)
  BaseTypeIsReadOnly = 0
  BaseType = LinearPeriodic
    MeasurementUnit = 5066068
    MeasurementResolutionIsReadOnly = 0
    MeasurementResolution = 0.01
    CountDirectionIsReadOnly = 0
    CountDirection = Standard
    PeriodSettings:
      Period = 2000
  MovementLimitsIsReadOnly = 0
  MovementLimits = Internal
    Position:
      LowerLimitMin = -1.79769313486231E308
      UpperLimitMax = 1.79769313486231E308
      LowerLimit = -1000.0
      UpperLimit = 1000.0
    VelocityIsReadOnly = 0
    Velocity:
      VelocityMax = 3.4E38
      Velocity = 2000
    AccelerationIsReadOnly = 0
    Acceleration:
      AccelerationMax = 3.4E38
      Acceleration = 100
    DecelerationIsReadOnly = 0
    Deceleration:
      DecelerationMax = 3.4E38
      Deceleration = 100
  Alarms = None
```

### Config_6.axesgroupfeature - 5APC3100_KBU1_000/mappMotion/Config_6.axesgroupfeature
```
Element Feature_FrameHierarchy (Type=axesgroupfeature)
  Type = FrameHierarchy
    ModalDataBehaviour = UseAxesGroupSettings
    FrameHierarchy = Custom
      FramePropertyMapping:
        BCS = RoboBase
        PCS = ZeroPosPickConveyor
        SCS1
        SCS2
        SCS3
        SCS4
        SCS5
      MCS:
        Name = MachineBase
        Frame[1]:
          Name = RoboBase
          Type = StandardFrame
            Translation:
              X = 0.0
              Y = 0.0
              Z = 490
            Orientation:
              Angle1 = 0.0
              Angle2 = 0.0
              Angle3 = 0.0
          Frame[1]:
            Name = ZeroPosPickConveyor
            Type = StandardFrame
              Translation:
                X = -300
                Y = 0
                Z = -430
              Orientation:
                Angle1 = 0.0
                Angle2 = 0.0
                Angle3 = 0.0
Element Feature_Tracking (Type=axesgroupfeature)
  Type = Tracking
    ModalDataBehaviour = UseAxesGroupSettings
    SynchronisationGeometry = Basic
      CartesianRadius = 20.0
    TorqueLimitConsideration = Exact
Element Feature_PathDefinition (Type=axesgroupfeature)
  Type = PathDefinitions
    ModalDataBehaviour = UseAxesGroupSettings
    PathDefinition[1]:
      Name = Path1
      Type = CartesianPath
        CalculatedIn = PCS
      Limit = Internal
        Velocity = NotUsed
        Acceleration = NotUsed
        Deceleration = NotUsed
        Jerk = NotUsed
```

### Config_7.pickobjectlist - 5APC3100_KBU1_000/mappMotion/Config_7.pickobjectlist
```
Element gPickObjectList_1 (Type=pickobjectlist)
  Object[1] = SingleItem
    Name = MyProduct
  Object[2] = Container
    Name = MyCont
    Layer[1]:
      Position[1]:
        Object = MyProduct
        Translation:
          X = 4
          Y = 0.0
          Z = 0.0
        Orientation:
          Angle1 = 0.0
          Angle2 = 0.0
          Angle3 = 0.0
      Position[2]:
        Object = MyProduct
        Translation:
          X = 48
          Y = 0.0
          Z = 0.0
        Orientation:
          Angle1 = 0.0
          Angle2 = 0.0
          Angle3 = 0.0
      Position[3]:
        Object = MyProduct
        Translation:
          X = 96
          Y = 0.0
          Z = 0.0
        Orientation:
          Angle1 = 0.0
          Angle2 = 0.0
          Angle3 = 0.0
      Position[4]:
        Object = MyProduct
        Translation:
          X = 144
          Y = 0.0
          Z = 0.0
        Orientation:
          Angle1 = 0.0
          Angle2 = 0.0
          Angle3 = 0.0
```

### Config_8.pickregister - 5APC3100_KBU1_000/mappMotion/Config_8.pickregister
```
Element gPickRegister (Type=pickregister)
  Type = LinearConveyor
    StandardFrameName = ConveyorPick
    Length = 600
    Width = 120
    Height = 6
    MaxPositionError = 10
    MotionSource = Axis
      AxisRef = gAxis_1
      MovementLimits = UseAxisLimits
        Direction = Bidirectional
  SceneViewerObject = Used
    VisualRepresentation = Conveyor belt
      Dimensions:
        Length = 0.0
        Width = 0.0
        Height = 0.0
      Translation:
        X = 0.0
        Y = 0.0
        Z = 0.0
      Orientation:
        Angle1 = 0.0
        Angle2 = 0.0
        Angle3 = 0.0
    Content:
      Template[1]:
        VisualRepresentation = 2DShape
          ShapeType:
            Dimensions:
              Radius = 25.0
            Translation:
              X = 0.0
              Y = 0.0
              Z = 0.0
            Orientation:
              Angle1 = 0.0
              Angle2 = 0.0
              Angle3 = 0.0
        Filter:
          ObjectState:
            State[1] = 1
      Template[2]:
        VisualRepresentation:
          Size = 50.0
        Filter:
          ObjectState:
            State[1] = 2
  Alarms = None
Element gPlaceRegister (Type=pickregister)
  Type = LinearConveyor
    StandardFrameName = ConveyorPlace
    Length = 215
    Width = 60
    Height = 10
    MaxItems = 5
    MaxPositionError = 10
    MotionSource = Axis
      AxisRef = gAxis_2
      MovementLimits = UseAxisLimits
        Direction = Bidirectional
  SceneViewerObject = Used
    VisualRepresentation = Cuboid
      Dimensions:
        Length = 215
        Width = 60
        Height = 50
      Translation:
        X = 0.0
        Y = 0.0
        Z = 0.0
      Orientation:
        Angle1 = 0.0
        Angle2 = 0.0
        Angle3 = 0.0
    Content:
      Template[1]:
        VisualRepresentation = 2DShape
          ShapeType:
            Dimensions:
              Radius = 25.0
            Translation:
              X = 0.0
              Y = 0.0
              Z = 0.0
            Orientation:
              Angle1 = 0.0
              Angle2 = 0.0
              Angle3 = 0.0
        Filter:
          ObjectState:
            State[1] = 1
      Template[2]:
        VisualRepresentation:
          Size = 50.0
        Filter:
          ObjectState:
            State[1] = 1
  Alarms = MpAlarmX
```

### Config_9.pickcore - 5APC3100_KBU1_000/mappMotion/Config_9.pickcore
```
Element gPickCore_1 (Type=pickcore)
  AxesGroupRef = g4AxDeltaA
  Gripper = Standard
    Behavior:
      ProcessVariableName = ::PrgPickCor:Gripper
  Job[1]:
    JobName = PickToPlace
    Object = MyProduct
    InfeedRegister = gPickRegister
    OutfeedRegister = gPlaceRegister
    Movement = Basic
      PickOffsetZ = 20
      PickRounding = 10
      PlaceOffsetZ = 20
      PlaceRounding = 10
    Limits = Basic
      WithObject:
        Velocity = 700
        Acceleration = 2000
        Deceleration = 2000
      WithoutObject:
        Velocity = 700
        Acceleration = 2000
        Deceleration = 2000
  OperationMode[1]:
    Name = ConveyorToConveyor
    AssignedJob[1]:
      Name = PickToPlace
      Processing = FIFO
      JobExecBehav = WaitForPlaceHolder
    AssignedJob[2]:
      Name
      Processing = FIFO
      JobExecBehav = WaitForPlaceHolder
    AssignedJob[3]:
      Name
      Processing = FIFO
      JobExecBehav = WaitForPlaceHolder
    AssignedJob[4]:
      Name
      Processing = FIFO
      JobExecBehav = WaitForPlaceHolder
    AssignedJob[5]:
      Name
      Processing = FIFO
      JobExecBehav = WaitForPlaceHolder
    AssignedJob[6]:
      Name
      Processing = FIFO
      JobExecBehav = WaitForPlaceHolder
    AssignedJob[7]:
      Name
      Processing = FIFO
      JobExecBehav = WaitForPlaceHolder
    AssignedJob[8]:
      Name
      Processing = FIFO
      JobExecBehav = WaitForPlaceHolder
    AssignedJob[9]:
      Name
      Processing = FIFO
      JobExecBehav = WaitForPlaceHolder
    AssignedJob[10]:
      Name
      Processing = FIFO
      JobExecBehav = WaitForPlaceHolder
    IdleBehavior = StayFixedWaitingPosition
      Position:
        StandardFrameName = PnPWaitingPosition
        Translation:
          X = 0.0
          Y = 0.0
          Z = 0.0
        Orientation:
          Angle1 = 0.0
          Angle2 = 0.0
          Angle3 = 0.0
  Alarms = MpAlarmX
```

### Config_13.mpalarmxcore - 5APC3100_KBU1_000/mappServices/Config_13.mpalarmxcore
```
Element gAlarmXCore (Type=mpalarmxcore)
  mapp.AlarmX.Core.Configuration:
    [0]:
      Name = PickCoreError
      Message = {$AlarmText/PickCoreError}
      Code = 1
      Severity = 10
      Behavior = PersistentAlarm
    [1]:
      Name = PickRegisterError
      Message = {$AlarmText/PickRegisterError}
      Code = 2
      Severity = 10
      Behavior = PersistentAlarm
    [2]:
      Name = PlaceRegisterError
      Message = {$AlarmText/PlaceRegisterError}
      Code = 3
      Severity = 10
      Behavior = PersistentAlarm
    [3]:
      Name = ConveyorAxisError
      Message = {$AlarmText/ConveyorAxisError}
      Code = 4
      Severity = 10
      Behavior = PersistentAlarm
    [4]:
      Name = ConveyorVirtualAxisError
      Message = {$AlarmText/ConveyorVirtualAxis}
      Code = 5
      Severity = 10
      Behavior = PersistentAlarm
    [5]:
      Name = DeltaVirtualAxisError
      Message = {$AlarmText/DeltaVirtualAxisError}
      Code = 6
      Severity = 10
      Behavior = PersistentAlarm
    [6]:
      Name = DeltaAxis1Error
      Message = {$AlarmText/DeltaAxis1Error}
      Code = 7
      Severity = 10
      Behavior = PersistentAlarm
    [7]:
      Name = DeltaAxis2Error
      Message = {$AlarmText/DeltaAxis2Error}
      Code = 8
      Severity = 10
      Behavior = PersistentAlarm
    [8]:
      Name = DeltaAxis3Error
      Message = {$AlarmText/DeltaAxis3Error}
      Code = 9
      Severity = 10
      Behavior = PersistentAlarm
    [9]:
      Name = DeltaError
      Message = {$AlarmText/DeltaError}
      Code = 10
      Severity = 10
      Behavior = PersistentAlarm
    [10]:
      Name = PickRegCreateProductError
      Message = {$AlarmText/PickRegCreate}
      Code = 11
      Severity = 10
      Behavior = PersistentAlarm
  mapp.AlarmX.Core.Snippets:
    [0]:
      Key = 
```

### Config_1.axesgroup - X20CP0484_1/mappMotion/3AxesDeltaA/Config_1.axesgroup
```
Element g3AxDeltaA (Type=axesgroup)
  Type = PathGenAxesGroup
    ProcessingTaskClass = 255
    License = 1
    PhysicalAxes:
      JointAxes:
        JointAxisAxisRefIsReadOnly = 0
        JointAxis[1]:
          Name = Q1
          AxisRef = gAxisQ1
        JointAxis[2]:
          Name = Q2
          AxisRef = gAxisQ2
        JointAxis[3]:
          Name = Q3
          AxisRef = gAxisQ3
    MechanicalSystem:
      MechSysRefIsReadOnly = 0
      MechSysRef = MechSys_3AxDeltaA
    BasicSettings:
      ModalDataBehaviour = ResetToDefault
      GeometryPlanning:
        TCPResolutionIsReadOnly = 0
        TCPResolution:
          LengthResolution = 0.001
          AngleResolution = 0.001
        Rounding:
          PathDistance = 0.0
          SymmetricRounding = Yes
          LastSegment = Half
          AvoidZeroCurvature = No
        RoundingMode = Standard
        MaxCornerDeviation = 0.0
        MaxTangentialTransitionDeviation = 0.0
        MaxRadiusDeviation = 0.001
        WorkingPlane = XY
      TrajectoryPlanningIsReadOnly = 0
      TrajectoryPlanning = Basic
        LimitCheckResolutionIsReadOnly = 0
        LimitCheckResolution = UserDefinedTime
          TimeIsReadOnly = 0
          Time = 0.01
        BufferTime = UserDefinedTime
          Time = 0.1
        BarrierParametrization = JointCoordinates
        TorqueLimitConsideration = Exact
      Miscellaneous:
        NonMovementsLimit = NotUsed
        TimeStretchOverride:
          JerkSuppression = NotUsed
    StopReaction:
      AxisError:
        AxisReactionIsReadOnly = 0
    AxesGroupFeatures:
      FeatureRef[1] = Feature_Programs
      FeatureRef[2] = Feature_Jogging
  Alarms = None
```

### Config_2.axis - X20CP0484_1/mappMotion/3AxesDeltaA/Config_2.axis
```
Element gAxisQ1 (Type=axis)
  BaseTypeIsReadOnly = 0
  BaseType = RotaryBounded
    MeasurementUnitIsReadOnly = 0
    MeasurementUnit = 17476
    MeasurementResolutionIsReadOnly = 0
    MeasurementResolution = 0.01
    CountDirectionIsReadOnly = 0
    CountDirection = Standard
  MovementLimitsIsReadOnly = 0
  MovementLimits = Internal
    Position:
      LowerLimitMin = -1.79769313486231E308
      UpperLimitMax = 1.79769313486231E308
      LowerLimit = -1000.0
      UpperLimit = 1000.0
    VelocityIsReadOnly = 0
    Velocity:
      VelocityMax = 3.4E38
      Velocity = 10.0
    AccelerationIsReadOnly = 0
    Acceleration:
      AccelerationMax = 3.4E38
      Acceleration = 50.0
    DecelerationIsReadOnly = 0
    Deceleration:
      DecelerationMax = 3.4E38
      Deceleration = 50.0
  Alarms = None
Element gAxisQ2 (Type=axis)
  BaseTypeIsReadOnly = 0
  BaseType = RotaryBounded
    MeasurementUnitIsReadOnly = 0
    MeasurementUnit = 17476
    MeasurementResolutionIsReadOnly = 0
    MeasurementResolution = 0.01
    CountDirectionIsReadOnly = 0
    CountDirection = Standard
  MovementLimitsIsReadOnly = 0
  MovementLimits = Internal
    Position:
      LowerLimitMin = -1.79769313486231E308
      UpperLimitMax = 1.79769313486231E308
      LowerLimit = -1000.0
      UpperLimit = 1000.0
    VelocityIsReadOnly = 0
    Velocity:
      VelocityMax = 3.4E38
      Velocity = 10.0
    AccelerationIsReadOnly = 0
    Acceleration:
      AccelerationMax = 3.4E38
      Acceleration = 50.0
    DecelerationIsReadOnly = 0
    Deceleration:
      DecelerationMax = 3.4E38
      Deceleration = 50.0
  Alarms = None
Element gAxisQ3 (Type=axis)
  BaseTypeIsReadOnly = 0
  BaseType = RotaryBounded
    MeasurementUnitIsReadOnly = 0
    MeasurementUnit = 17476
    MeasurementResolutionIsReadOnly = 0
    MeasurementResolution = 0.01
    CountDirectionIsReadOnly = 0
    CountDirection = Standard
  MovementLimitsIsReadOnly = 0
  MovementLimits = Internal
    Position:
      LowerLimitMin = -1.79769313486231E308
      UpperLimitMax = 1.79769313486231E308
      LowerLimit = -1000.0
      UpperLimit = 1000.0
    VelocityIsReadOnly = 0
    Velocity:
      VelocityMax = 3.4E38
      Velocity = 10.0
    AccelerationIsReadOnly = 0
    Acceleration:
      AccelerationMax = 3.4E38
      Acceleration = 50.0
    DecelerationIsReadOnly = 0
    Deceleration:
      DecelerationMax = 3.4E38
      Deceleration = 50.0
  Alarms = None
```

### Config_3.mechanicalsystem - X20CP0484_1/mappMotion/3AxesDeltaA/Config_3.mechanicalsystem
```
Element MechSys_3AxDeltaA (Type=mechanicalsystem)
  TypeIsReadOnly = 0
  Type = Delta
    SubtypeIsReadOnly = 0
    Subtype = 3AxesDeltaA
      SceneViewerObject = Generic
      DescriptionIsReadOnly = 0
      Description = Standard
        Dimensions:
          BasePlatform:
            CenterIsReadOnly = 0
            Center:
              X = 0.0
              Y = 0.0
              Z = 0.0
            ArmLinkPointIsReadOnly = 0
            Arm1LinkPoint:
              Angle = 0.0
              Radius = 250.0
              Z = 0.0
            Arm2LinkPoint:
              Angle = 120.0
              Radius = 250.0
              Z = 0.0
            Arm3LinkPoint:
              Angle = 240.0
              Radius = 250.0
              Z = 0.0
          Arms:
            ArmIsReadOnly = 0
            Arm1:
              UpperArmLength = 600.0
              LowerArmLength = 900.0
            Arm2:
              UpperArmLength = 600.0
              LowerArmLength = 900.0
            Arm3:
              UpperArmLength = 600.0
              LowerArmLength = 900.0
            LowerArmPairDistance = 0.0
          EndEffectorPlatform:
            ArmLinkPointIsReadOnly = 0
            Arm1LinkPoint:
              Radius = 50.0
              Z = 0.0
            Arm2LinkPoint:
              Radius = 50.0
              Z = 0.0
            Arm3LinkPoint:
              Radius = 50.0
              Z = 0.0
            TranslationToFlangeIsReadOnly = 0
            TranslationToFlange:
              X = 0.0
              Y = 0.0
              Z = -150
        Offsets:
          JointAxisIsReadOnly = 0
          JointAxis[1] = 0.0
          JointAxis[2] = 0.0
          JointAxis[3] = 0.0
        CountDirections:
          JointAxisIsReadOnly = 0
          JointAxis[1] = Standard
          JointAxis[2] = Standard
          JointAxis[3] = Standard
      CoordinatesNames = Default
        XCoordinateName = X
        YCoordinateName = Y
        ZCoordinateName = Z
      WireFrameModelIsReadOnly = 0
      WireFrameModel = Standard
        UpperArm1IsReadOnly = 0
        UpperArm1 = ConnectionLine
          DistanceMin = -1.79769313486231E308
          DistanceMax = 1.79769313486231E308
          Distance = 0.0
        LowerArm1IsReadOnly = 0
        LowerArm1 = ConnectionLine
          DistanceMin = -1.79769313486231E308
          DistanceMax = 1.79769313486231E308
          Distance = 0.0
        UpperArm2IsReadOnly = 0
        UpperArm2 = ConnectionLine
          DistanceMin = -1.79769313486231E308
          DistanceMax = 1.79769313486231E308
          Distance = 0.0
        LowerArm2IsReadOnly = 0
        LowerArm2 = ConnectionLine
          DistanceMin = -1.79769313486231E308
          DistanceMax = 1.79769313486231E308
          Distance = 0.0
        UpperArm3IsReadOnly = 0
        UpperArm3 = ConnectionLine
          DistanceMin = -1.79769313486231E308
          DistanceMax = 1.79769313486231E308
          Distance = 0.0
        LowerArm3IsReadOnly = 0
        LowerArm3 = ConnectionLine
          DistanceMin = -1.79769313486231E308
          DistanceMax = 1.79769313486231E308
          Distance = 0.0
        EndEffectorPlatformToFlangeIsReadOnly = 0
        EndEffectorPlatformToFlange = ConnectionLine
          DistanceMin = -1.79769313486231E308
          DistanceMax = 1.79769313486231E308
          Distance = 0.0
        FlangeToTcp = ConnectionLine
          DistanceMin = -1.79769313486231E308
          DistanceMax = 1.79769313486231E308
          Distance = 0.0
      DynamicModelIsReadOnly = 0
      DynamicModel = DynParTable
        TableRef
      InternalDynamicModelIsReadOnly = 0
      InternalDynamicModel = NotUsed
      DynamicLimits = DynParTables
        GearboxLimitsTableRef
        CrossSectionLimitsTableRef
      InternalDynamicLimits = NotUsed
      LoadDependentJerkLimitsIsReadOnly = 0
      LoadDependentJerkLimits = NotUsed
      CouplingsIsInvisible = 0
      JointAxesPositionLimits:
        JointAxisIsReadOnly = 0
        JointAxis[1] = UseAxisLimits
        JointAxis[2] = UseAxisLimits
        JointAxis[3] = UseAxisLimits
```

### Config_11.axis - X20CP0484_1/mappMotion/4AxesDeltaA/Config_11.axis
```
Element gAxisQ1 (Type=axis)
  BaseTypeIsReadOnly = 0
  BaseType = RotaryBounded
    MeasurementUnitIsReadOnly = 0
    MeasurementUnit = 17476
    MeasurementResolutionIsReadOnly = 0
    MeasurementResolution = 0.01
    CountDirectionIsReadOnly = 0
    CountDirection = Standard
  MovementLimitsIsReadOnly = 0
  MovementLimits = Internal
    Position:
      LowerLimitMin = -1.79769313486231E308
      UpperLimitMax = 1.79769313486231E308
      LowerLimit = -1000.0
      UpperLimit = 1000.0
    VelocityIsReadOnly = 0
    Velocity:
      VelocityMax = 3.4E38
      Velocity = 10.0
    AccelerationIsReadOnly = 0
    Acceleration:
      AccelerationMax = 3.4E38
      Acceleration = 50.0
    DecelerationIsReadOnly = 0
    Deceleration:
      DecelerationMax = 3.4E38
      Deceleration = 50.0
  Alarms = None
Element gAxisQ2 (Type=axis)
  BaseTypeIsReadOnly = 0
  BaseType = RotaryBounded
    MeasurementUnitIsReadOnly = 0
    MeasurementUnit = 17476
    MeasurementResolutionIsReadOnly = 0
    MeasurementResolution = 0.01
    CountDirectionIsReadOnly = 0
    CountDirection = Standard
  MovementLimitsIsReadOnly = 0
  MovementLimits = Internal
    Position:
      LowerLimitMin = -1.79769313486231E308
      UpperLimitMax = 1.79769313486231E308
      LowerLimit = -1000.0
      UpperLimit = 1000.0
    VelocityIsReadOnly = 0
    Velocity:
      VelocityMax = 3.4E38
      Velocity = 10.0
    AccelerationIsReadOnly = 0
    Acceleration:
      AccelerationMax = 3.4E38
      Acceleration = 50.0
    DecelerationIsReadOnly = 0
    Deceleration:
      DecelerationMax = 3.4E38
      Deceleration = 50.0
  Alarms = None
Element gAxisQ3 (Type=axis)
  BaseTypeIsReadOnly = 0
  BaseType = RotaryBounded
    MeasurementUnitIsReadOnly = 0
    MeasurementUnit = 17476
    MeasurementResolutionIsReadOnly = 0
    MeasurementResolution = 0.01
    CountDirectionIsReadOnly = 0
    CountDirection = Standard
  MovementLimitsIsReadOnly = 0
  MovementLimits = Internal
    Position:
      LowerLimitMin = -1.79769313486231E308
      UpperLimitMax = 1.79769313486231E308
      LowerLimit = -1000.0
      UpperLimit = 1000.0
    VelocityIsReadOnly = 0
    Velocity:
      VelocityMax = 3.4E38
      Velocity = 10.0
    AccelerationIsReadOnly = 0
    Acceleration:
      AccelerationMax = 3.4E38
      Acceleration = 50.0
    DecelerationIsReadOnly = 0
    Deceleration:
      DecelerationMax = 3.4E38
      Deceleration = 50.0
  Alarms = None
Element gAxisQ4 (Type=axis)
  BaseTypeIsReadOnly = 0
  BaseType = Rotary
    MeasurementUnitIsReadOnly = 0
    MeasurementUnit = 17476
    MeasurementResolutionIsReadOnly = 0
    MeasurementResolution = 0.01
    CountDirectionIsReadOnly = 0
    CountDirection = Standard
  MovementLimitsIsReadOnly = 0
  MovementLimits = Internal
    Position:
      LowerLimitMin = -1.79769313486231E308
      UpperLimitMax = 1.79769313486231E308
      LowerLimit = -1000.0
      UpperLimit = 1000.0
    VelocityIsReadOnly = 0
    Velocity:
      VelocityMax = 3.4E38
      Velocity = 10.0
    AccelerationIsReadOnly = 0
    Acceleration:
      AccelerationMax = 3.4E38
      Acceleration = 50.0
    DecelerationIsReadOnly = 0
    Deceleration:
      DecelerationMax = 3.4E38
      Deceleration = 50.0
  Alarms = None
```

### Config_14.axis - X20CP0484_1/mappMotion/Config_14.axis
```
Element gAxis_1 (Type=axis)
  BaseTypeIsReadOnly = 0
  BaseType = LinearPeriodic
    MeasurementUnit = 5066068
    MeasurementResolutionIsReadOnly = 0
    MeasurementResolution = 0.01
    CountDirectionIsReadOnly = 0
    CountDirection = Standard
    PeriodSettings:
      Period = 2000
  MovementLimitsIsReadOnly = 0
  MovementLimits = Internal
    Position:
      LowerLimitMin = -1.79769313486231E308
      UpperLimitMax = 1.79769313486231E308
      LowerLimit = -1000.0
      UpperLimit = 1000.0
    VelocityIsReadOnly = 0
    Velocity:
      VelocityMax = 3.4E38
      Velocity = 100
    AccelerationIsReadOnly = 0
    Acceleration:
      AccelerationMax = 3.4E38
      Acceleration = 10
    DecelerationIsReadOnly = 0
    Deceleration:
      DecelerationMax = 3.4E38
      Deceleration = 10
  Alarms = None
Element gAxis_2 (Type=axis)
  BaseTypeIsReadOnly = 0
  BaseType = LinearPeriodic
    MeasurementUnit = 5066068
    MeasurementResolutionIsReadOnly = 0
    MeasurementResolution = 0.01
    CountDirectionIsReadOnly = 0
    CountDirection = Standard
    PeriodSettings:
      Period = 2000
  MovementLimitsIsReadOnly = 0
  MovementLimits = Internal
    Position:
      LowerLimitMin = -1.79769313486231E308
      UpperLimitMax = 1.79769313486231E308
      LowerLimit = -1000.0
      UpperLimit = 1000.0
    VelocityIsReadOnly = 0
    Velocity:
      VelocityMax = 3.4E38
      Velocity = 100
    AccelerationIsReadOnly = 0
    Acceleration:
      AccelerationMax = 3.4E38
      Acceleration = 10
    DecelerationIsReadOnly = 0
    Deceleration:
      DecelerationMax = 3.4E38
      Deceleration = 10
  Alarms = None
```

### Config_6.axesgroupfeature - X20CP0484_1/mappMotion/Config_6.axesgroupfeature
```
Element Feature_FrameHierarchy (Type=axesgroupfeature)
  Type = FrameHierarchy
    ModalDataBehaviour = UseAxesGroupSettings
    FrameHierarchy = Custom
      FramePropertyMapping:
        BCS = RoboBase
        PCS = ZeroPosPickConveyor
        SCS1
        SCS2
        SCS3
        SCS4
        SCS5
      MCS:
        Name = MachineBase
        Frame[1]:
          Name = RoboBase
          Type = StandardFrame
            Translation:
              X = 0.0
              Y = 0.0
              Z = 1000
            Orientation:
              Angle1 = 0.0
              Angle2 = 0.0
              Angle3 = 0.0
          Frame[1]:
            Name = ZeroPosPickConveyor
            Type = StandardFrame
              Translation:
                X = 0.0
                Y = 400
                Z = -1000
              Orientation:
                Angle1 = 0.0
                Angle2 = 0.0
                Angle3 = 0.0
Element Feature_Tracking (Type=axesgroupfeature)
  Type = Tracking
    ModalDataBehaviour = UseAxesGroupSettings
    SynchronisationGeometry = Basic
      CartesianRadius = 20.0
Element Feature_PathDefinition (Type=axesgroupfeature)
  Type = PathDefinitions
    ModalDataBehaviour = UseAxesGroupSettings
    PathDefinition[1]:
      Name = Path1
      Type = CartesianPath
        CalculatedIn = PCS
      Limit = Internal
        Velocity = NotUsed
        Acceleration = NotUsed
        Deceleration = NotUsed
        Jerk = NotUsed
```

### Config_8.pickregister - X20CP0484_1/mappMotion/Config_8.pickregister
```
Element gPickRegister (Type=pickregister)
  Type = LinearConveyor
    StandardFrameName = ConveyorPick
    Length = 2000
    Width = 250
    Height = 100
    MotionSource = Axis
      AxisRef = gAxis_1
      MovementLimits = UseAxisLimits
        Direction = Bidirectional
  SceneViewerObject = Used
    Content:
      Template[1]:
        VisualRepresentation:
          Size = 50.0
  Alarms = None
Element gPlaceRegister (Type=pickregister)
  Type = LinearConveyor
    StandardFrameName = ConveyorPlace
    Length = 2000
    Width = 250.0
    Height = 100
    MotionSource = Axis
      AxisRef = gAxis_2
      MovementLimits = UseAxisLimits
        Direction = Bidirectional
  SceneViewerObject = Used
    Content:
      Template[1]:
        VisualRepresentation:
          Size = 50.0
  Alarms = None
```

## Logical view

Binary libraries used (declarations not repeated): operator, runtime, astime, AsIecCon, AsZip, FileIO, Library, AsARCfg, powerlnk, AsEPL, AsIO, sys_lib, DataObj, McBase, MpBase, McTrkPath, McPathGen, MpAxis, McPureVAx, MpPick, McAcpAx, McAxis, McProgInt, McAxGroup, MpRobotics, ViBase 5.26.1, CoTrace, MpAlarmX

### Global.var - Global variables
```iecst
VAR
	iloscMonet : UDINT;
END_VAR
```

### Package Logical/Libraries - Global libraries

### PrgGlobal.var - Pick and place global variables
```iecst
VAR
	Mode : BOOL := TRUE;
	restart : BOOL;
	CmdStart : BOOL := FALSE; (*Set = 1 to start the process*)
	ReadyMechanics : BOOL := FALSE;
	ReadyPickCore : BOOL := FALSE;
	ReadyPickReg : BOOL := FALSE;
	ReadyPlaceReg : BOOL := FALSE;
	ReadyToStart : BOOL := FALSE;
	PickConveyorPosition : LREAL;
	PickConveyorLength : LREAL := 600; (*must be the same as pick conveyor length in MpPick configuration*)
	PlaceConveyorPosition : LREAL;
	PlaceConveyorLength : LREAL := 215; (*must be the same as place conveyor length in MpPick configuration*)
	setZ : LREAL;
	setY : LREAL;
	setX : LREAL;
	saveChanges : BOOL := FALSE;
	setAxis1 : LREAL;
	setAxis2 : LREAL;
	setAxis3 : LREAL;
	TCP : BOOL := TRUE;
	Gripper : BOOL;
END_VAR
```

### Program Logical/PickAndPlace/PrgMechs (IEC) - Handle Delta & Conveyor Belts

#### Variables.var
```iecst
VAR
	RC_Step : RCStepEnum;
	LastStep : RCStepEnum;
	MpDelta4Axis_0 : MpDelta4Axis;
	DeltaParameters : MpDelta4AxisParType;
	MpAxisBasic_0 : MpAxisBasic;
	AxisParameters_0 : MpAxisBasicParType;
	MpAxisBasic_1 : MpAxisBasic;
	AxisParameters_1 : MpAxisBasicParType;
	FB_AlarmHistory : MpAlarmXHistory;
	FB_AlarmCore : MpAlarmXCore;
END_VAR
```

#### Main.st
```iecst
PROGRAM _INIT

	MpDelta4Axis_0.Override := 100.0;
	MpDelta4Axis_0.Enable   := TRUE;

	AxisParameters_0.Velocity     := 50.0;
	AxisParameters_0.Acceleration := 50.0;
	AxisParameters_0.Deceleration := 50.0;

	AxisParameters_1.Velocity     := 130.0;
	AxisParameters_1.Acceleration := 50.0;
	AxisParameters_1.Deceleration := 50.0;

	MpAxisBasic_0.Enable := TRUE;
	MpAxisBasic_1.Enable := TRUE;

	FB_AlarmCore.MpLink := ADR(gAlarmXCore);
	FB_AlarmCore.Enable := TRUE;
	FB_AlarmHistory.MpLink := ADR(gAlarmXHistory);
	FB_AlarmHistory.Enable := TRUE;

	// dummy call of axis PVs just to avoid warning -2141192189 "The PV 'gAxisQx' does not exists" in logger
	gAxisQ1;
	gAxisQ2;
	gAxisQ3;
	gAxisQ4;

END_PROGRAM

PROGRAM _CYCLIC

    (* Prepare mechanics: Robot & conveyors *)
	CASE RC_Step OF

		(* first preparing robot *)
		RC_WAIT_ENABLE:
			IF MpDelta4Axis_0.Active THEN
				RC_Step := RC_POWER_ROBOT;
			END_IF

		RC_POWER_ROBOT:
			MpDelta4Axis_0.Power := TRUE;
			IF MpDelta4Axis_0.PowerOn THEN
				RC_Step := RC_HOME_ROBOT;
			END_IF

		RC_HOME_ROBOT:
			MpDelta4Axis_0.Home := TRUE;
			IF MpDelta4Axis_0.IsHomed THEN
				MpDelta4Axis_0.Home := FALSE;
				RC_Step := RC_ROBOT_READY;
			END_IF

		RC_ROBOT_READY:
			RC_Step := RC_WAIT_ENABLE_AXIS_FB;

			(* preparing conveyors *)
		RC_WAIT_ENABLE_AXIS_FB:
			IF MpAxisBasic_0.Active THEN
				IF MpAxisBasic_1.Active THEN
					RC_Step := RC_POWER_AXIS;
				END_IF
			ELSIF MpAxisBasic_0.Error  THEN
				LastStep := RC_Step;
				RC_Step  := RC_ERROR;
			END_IF;

		RC_POWER_AXIS:
			MpAxisBasic_0.Power := TRUE;
			MpAxisBasic_1.Power := TRUE;
			RC_Step := RC_WAIT_POWER_AXIS;

		RC_WAIT_POWER_AXIS:
			IF MpAxisBasic_0.PowerOn THEN
				IF MpAxisBasic_1.PowerOn THEN
					RC_Step := RC_HOME_AXIS;
				END_IF
			ELSIF MpAxisBasic_0.Error  THEN
				LastStep := RC_Step;
				RC_Step  := RC_ERROR;
			END_IF;

		RC_HOME_AXIS:
			MpAxisBasic_0.Home := TRUE;
			MpAxisBasic_1.Home := TRUE;
			RC_Step := RC_WAIT_HOME_AXIS;

		RC_WAIT_HOME_AXIS:
			IF MpAxisBasic_0.IsHomed THEN
				IF MpAxisBasic_0.IsHomed THEN
					MpAxisBasic_0.Home := FALSE;
					MpAxisBasic_1.Home := FALSE;
					RC_Step := RC_READY;
				END_IF
			ELSIF MpAxisBasic_0.Error  THEN
				LastStep := RC_Step;
				RC_Step  := RC_ERROR;
			END_IF;

		RC_READY:
			ReadyMechanics := TRUE;
			IF CmdStart AND ReadyToStart THEN
				RC_Step := RC_START_PROCESS;
			END_IF;

			(* start conveyors to move *)
		RC_START_PROCESS:
			MpAxisBasic_0.MoveVelocity := TRUE;
			//  MpAxisBasic_1.MoveVelocity := TRUE;
			RC_Step := RC_WAIT_PROCESS_STARTED;

		RC_WAIT_PROCESS_STARTED:
			IF MpAxisBasic_0.Info.PLCopenState = mcAXIS_CONTINUOUS_MOTION THEN
				//   IF MpAxisBasic_1.Info.PLCopenState = mcAXIS_CONTINUOUS_MOTION THEN
				RC_Step := RC_PROCESSING;
				//  END_IF
			ELSIF MpAxisBasic_0.Error  THEN
				LastStep := RC_Step;
				RC_Step  := RC_ERROR;
			END_IF;

		RC_PROCESSING:
			IF MpAxisBasic_0.Error  THEN
				LastStep := RC_Step;
				RC_Step  := RC_ERROR;
			END_IF;

		RC_ERROR:
			ReadyMechanics := FALSE;

	END_CASE

	ReadyToStart := ReadyMechanics AND ReadyPickReg AND ReadyPlaceReg AND ReadyPickCore;

	IF MpDelta4Axis_0.Error THEN
		MpAlarmXSet(gAlarmXCore,'DeltaError');
	ELSE
		MpAlarmXReset(gAlarmXCore,'DeltaError');
	END_IF;

	IF MpAxisBasic_0.Error THEN
		MpAlarmXSet(gAlarmXCore,'ConveyorAxisError');
	ELSE
		MpAlarmXReset(gAlarmXCore,'ConveyorAxisError');
	END_IF;

	IF MpAxisBasic_1.Error THEN
		MpAlarmXSet(gAlarmXCore,'ConveyorVirtualAxisError');
	ELSE
		MpAlarmXReset(gAlarmXCore,'ConveyorVirtualAxisError');
	END_IF;

	(* Call FBs *)
	MpDelta4Axis_0.MpLink     := ADR(g4AxDeltaA);
	MpDelta4Axis_0.Parameters := ADR(DeltaParameters);
	MpDelta4Axis_0();

	MpAxisBasic_0.MpLink     := ADR(gAxis_1);
	MpAxisBasic_0.Parameters := ADR(AxisParameters_0);
	MpAxisBasic_0();

	MpAxisBasic_1.MpLink     := ADR(gAxis_2);
	MpAxisBasic_1.Parameters := ADR(AxisParameters_1);
	MpAxisBasic_1();

	PickConveyorPosition  := MpAxisBasic_0.Position;
	PlaceConveyorPosition := MpAxisBasic_1.Position;

END_PROGRAM
```

### Program Logical/PickAndPlace/PrgPickCore (IEC) - PickCore process handling

#### Variables.var
```iecst
VAR
	MpPickCore_0 : MpPickCore;
	LastStep : PickCoreStepEnum;
	PC_Step : PickCoreStepEnum;
	Error : BOOL;
END_VAR
```

#### Main.st
```iecst
PROGRAM _INIT

	PC_Step := PC_ENABLE_PICK_CORE;
	Gripper := FALSE;

END_PROGRAM

PROGRAM _CYCLIC

	CASE PC_Step OF

		(* Enable the PickCore *)
		PC_ENABLE_PICK_CORE:
			MpPickCore_0.Enable := TRUE;
			PC_Step := PC_WAIT_ENABLE_PICK_CORE;

		PC_WAIT_ENABLE_PICK_CORE:
			IF MpPickCore_0.Active THEN
				PC_Step := PC_ENABLE_CORE_PROCESS;

			ELSIF MpPickCore_0.Error THEN
				LastStep := PC_Step;
				PC_Step  := PC_ERROR;

			END_IF;

		PC_ENABLE_CORE_PROCESS:
			MpPickCore_0.ProcessEnable := TRUE;
			PC_Step := PC_WAIT_ENABLE_CORE_PROCESS;

		PC_WAIT_ENABLE_CORE_PROCESS:
			IF MpPickCore_0.ProcessActive THEN
				PC_Step := PC_READY_TO_START;

			ELSIF MpPickCore_0.Error THEN
				LastStep := PC_Step;
				PC_Step  := PC_ERROR;

			END_IF

		PC_READY_TO_START:
			ReadyPickCore := TRUE;

			IF CmdStart THEN
				MpPickCore_0.Parameters.OperationMode := 'ConveyorToConveyor';
				MpPickCore_0.ProcessStart := TRUE;
				PC_Step := PC_WAIT_START_CORE_PROCESS;
			END_IF

		PC_WAIT_START_CORE_PROCESS:
			IF MpPickCore_0.ProcessRunning THEN
				PC_Step := PC_STARTED;

			ELSIF MpPickCore_0.Error THEN
				LastStep := PC_Step;
				PC_Step  := PC_ERROR;

			END_IF;

		PC_STARTED:
			(* Nothing to do here *)
			iloscMonet := MpPickCore_0.Info.ProcessedObjects;
			IF MpPickCore_0.Error THEN
				LastStep := PC_Step;
				PC_Step  := PC_ERROR;
			END_IF;

		PC_ERROR:
			Error := TRUE;
			ReadyPickCore := FALSE;

	END_CASE
	(* Call FBs *)
	MpPickCore_0.MpLink := ADR(gPickCore_1);
	MpPickCore_0();

END_PROGRAM
```

### Program Logical/PickAndPlace/PrgPick (IEC) - Pick the products

#### Types.typ
```iecst
TYPE
	ConvStepEnum :
		(
		C_WAIT_ENABLE,
		C_ENABLE_REGISTER_FB,
		C_WAIT_ENABLE_REGISTER_FB,
		C_ENABLE_REGISTER,
		C_WAIT_ENABLE_REGISTER,
		C_ENABLE_ADD_REGISTER_FBS,
		C_WAIT_ENABLE_ADD_REGISTER_FBS,
		C_WAIT_START_PROCESS,
		C_START_PROCESS,
		C_WAIT_PROCESS_STARTED,
		C_PROCESSING,
		C_ERROR
	);
END_TYPE
```

#### Variables.var
```iecst
VAR
	C_Step : ConvStepEnum;
	LastStep : ConvStepEnum;
	Error : BOOL;
	ProductSpacing : LREAL;
	LastProductConveyorPosition : LREAL;
	ElapsedDistance : LREAL;
END_VAR
(*  *)
(*Functionblocks*)
VAR
	MpPickRegister_0 : MpPickRegister;
	MpPickRegCreateProduct : MpPickRegCreateObject;
	product : BOOL;
	iteracje : USINT;
END_VAR
```

#### Main.st
```iecst
PROGRAM _INIT

	C_Step := C_WAIT_ENABLE;
	Error := FALSE;

	ProductSpacing := 120; // distance between two consecutive products

END_PROGRAM

PROGRAM _CYCLIC

	CASE C_Step OF
		C_WAIT_ENABLE:
			LastStep := C_WAIT_ENABLE;
			C_Step   := C_ENABLE_REGISTER_FB;

			(* Pick-and-Place register handling for Picking conveyor *)
		C_ENABLE_REGISTER_FB:
			MpPickRegister_0.Enable := TRUE;
			C_Step := C_WAIT_ENABLE_REGISTER_FB;

		C_WAIT_ENABLE_REGISTER_FB:
			IF MpPickRegister_0.Active THEN
				C_Step := C_ENABLE_REGISTER;
			ELSIF MpPickRegister_0.Error THEN
				LastStep := C_Step;
				C_Step   := C_ERROR;
			END_IF;

		C_ENABLE_REGISTER:
			MpPickRegister_0.RegisterEnable := TRUE;
			C_Step := C_WAIT_ENABLE_REGISTER;

		C_WAIT_ENABLE_REGISTER:
			IF MpPickRegister_0.RegisterActive THEN
				C_Step := C_ENABLE_ADD_REGISTER_FBS;
			ELSIF MpPickRegister_0.Error THEN
				LastStep := C_Step;
				C_Step   := C_ERROR;
			END_IF;

		C_ENABLE_ADD_REGISTER_FBS:
			MpPickRegCreateProduct.Enable := TRUE;
			C_Step := C_WAIT_ENABLE_ADD_REGISTER_FBS;

		C_WAIT_ENABLE_ADD_REGISTER_FBS:
			IF MpPickRegCreateProduct.Active THEN
				C_Step := C_WAIT_START_PROCESS;
			ELSIF MpPickRegCreateProduct.Error THEN
				LastStep := C_Step;
				C_Step   := C_ERROR;
			END_IF;

		C_WAIT_START_PROCESS: // waits user start command and conveyor moving
			ReadyPickReg := TRUE;
			IF CmdStart AND ReadyToStart AND (PickConveyorPosition > 0) THEN
				C_Step := C_PROCESSING;
			END_IF;

		C_PROCESSING: (* now create products on moving conveyor for picking *)

			IF restart THEN
				MpPickRegCreateProduct.Parameters.LatchedConveyor.Position:= PickConveyorPosition;
				MpPickRegCreateProduct.Parameters.Mode := mpPICK_CREATE_SINGLEITEM;
				MpPickRegCreateProduct.Parameters.ObjectTypeName := 'MyProduct';
				MpPickRegCreateProduct.Parameters.Translation.X  := 0;
				MpPickRegCreateProduct.Parameters.Translation.Y  := 60;
				MpPickRegCreateProduct.Parameters.Translation.Z  := 2;// in the middle of conveyor width
				MpPickRegCreateProduct.Create := TRUE;

				LastProductConveyorPosition := MpPickRegCreateProduct.Parameters.LatchedConveyor.Position;
				restart :=0;
			ELSE
				MpPickRegCreateProduct.Create := FALSE;
			END_IF

			IF MpPickRegCreateProduct.Error THEN
				LastStep := C_Step;
				C_Step   := C_ERROR;
			END_IF;

		C_ERROR:
			Error := TRUE;
			ReadyPickReg := FALSE;

	END_CASE

	(* FB calls *)
	MpPickRegister_0.MpLink := ADR(gPickRegister);
	MpPickRegister_0();

	MpPickRegCreateProduct.MpLink := ADR(gPickRegister);
	MpPickRegCreateProduct();

END_PROGRAM
```

### Program Logical/PickAndPlace/PrgPlace (IEC) - Place the products

#### Variables.var
```iecst
VAR
	GetObjects1 : MpPickRegGetObjects;
	P_Step : PlaceStepEnum;
	LastStep : PlaceStepEnum;
	Error : BOOL;
	PlaceHoldersSpacing : LREAL;
	LastPlaceHolderConveyorPosition : LREAL;
	ElapsedDistance : LREAL;
END_VAR
(*   *)
(*Functionblocks*)
VAR
	MpPickRegCreatePlaceholder1 : MpPickRegCreateObject;
	MpPickRegCreatePlaceholder2 : MpPickRegCreateObject;
	MpPickRegCreatePlaceholder3 : MpPickRegCreateObject;
	MpPickRegCreatePlaceholder : MpPickRegCreateObject;
	MpPickRegister_0 : MpPickRegister;
	polka : USINT;
	tablicaPlace : ARRAY[0..3] OF LREAL;
	PlaceY : LREAL;
	iteracja : INT;
	MpPickRegCreateContainer : MpPickRegCreateObject;
	abc : BOOL := TRUE;
	ilosc1 : UINT;
	DeltaParameters : MpDelta4AxisParType;
	MpDelta4Axis_0 : MpDelta4Axis;
	AxisParam1 : MpAxisBasicParType;
	AxisParam2 : MpAxisBasicParType;
	AxisParam3 : MpAxisBasicParType;
	FB_Axis1 : MpAxisBasic;
	FB_Axis2 : MpAxisBasic;
	FB_Axis3 : MpAxisBasic;
	FB_Axis4 : MpAxisBasic;
	AxisParam4 : MpAxisBasicParType;
	tryb : BOOL;
	PHID : UDINT;
END_VAR
```

#### Main.st
```iecst
PROGRAM _INIT

	P_Step := P_WAIT_ENABLE;
	Error := FALSE;
	restart := FALSE;
	polka := 0;
	PlaceHoldersSpacing := 120; // distance between two consecutive place holders
	tablicaPlace[0] := 35;
	tablicaPlace[1] := 80;
	tablicaPlace[2] := 125;
	tablicaPlace[3] := 170;

	PlaceY := 30;

	abc := 0;
	iteracja := 0;
	tryb := 1;

END_PROGRAM

PROGRAM _CYCLIC

	CASE P_Step OF
		P_WAIT_ENABLE:
			P_Step := P_ENABLE_REGISTER_FB;

		P_ENABLE_REGISTER_FB:
			MpPickRegister_0.Enable := TRUE;
			P_Step := P_WAIT_ENABLE_REGISTER_FB;

		P_WAIT_ENABLE_REGISTER_FB:
			IF MpPickRegister_0.Active THEN
				P_Step := P_ENABLE_REGISTER_COMP;

			ELSIF MpPickRegister_0.Error THEN
				LastStep := P_Step;
				P_Step := P_ERROR;
			END_IF;

		P_ENABLE_REGISTER_COMP:
			MpPickRegister_0.RegisterEnable := TRUE;
			P_Step := P_WAIT_ENABLE_REGISTER_COMP;

		P_WAIT_ENABLE_REGISTER_COMP:
			IF MpPickRegister_0.RegisterActive THEN
				P_Step := P_ENABLE_ADD_REGISTER_FBS;

			ELSIF MpPickRegister_0.Error THEN
				LastStep := P_Step;
				P_Step := P_ERROR;
			END_IF;

		P_ENABLE_ADD_REGISTER_FBS:
			MpPickRegCreatePlaceholder.Enable := TRUE;
			MpPickRegCreatePlaceholder.Create := FALSE;
			P_Step := P_WAIT_ENABLE_ADD_REGISTER_FBS;

		P_WAIT_ENABLE_ADD_REGISTER_FBS:
			IF 	MpPickRegCreatePlaceholder.Active THEN
				P_Step := P_WAIT_START_PROCESS;

			ELSIF MpPickRegCreatePlaceholder.Error THEN
				LastStep := P_Step;
				P_Step := P_ERROR;
			END_IF;

		P_WAIT_START_PROCESS: // waits user start command and conveyor moving
			ReadyPlaceReg := TRUE;
			IF CmdStart AND ReadyToStart (*AND (PlaceConveyorPosition > 0)*) THEN
				P_Step := P_CREATE_OBJECTS;
			END_IF;

			(* We need to create positions (place holders) on place conveyor where to place picked objects *)
		P_CREATE_OBJECTS:

		//	IF tryb THEN

				IF abc THEN

					CASE iteracja OF
						0:
							MpPickRegCreatePlaceholder.Parameters.LatchedConveyor.Position := PlaceConveyorPosition;
							MpPickRegCreatePlaceholder.Parameters.Mode := mpPICK_CREATE_SINGLEITEM_PLACEH;
							MpPickRegCreatePlaceholder.Parameters.ObjectTypeName := 'MyProduct';
							MpPickRegCreatePlaceholder.Parameters.Translation.X := tablicaPlace[0];
							MpPickRegCreatePlaceholder.Parameters.Translation.Y := PlaceY; // in the middle of conveyor width
							MpPickRegCreatePlaceholder.Create := TRUE;
							PHID := MpPickRegCreatePlaceholder.ObjectPositionId;
							iteracja := 1;
							abc := 0;

						1:
							MpPickRegCreatePlaceholder.Parameters.LatchedConveyor.Position := PlaceConveyorPosition;
							MpPickRegCreatePlaceholder.Parameters.Mode := mpPICK_CREATE_SINGLEITEM_PLACEH;
							MpPickRegCreatePlaceholder.Parameters.ObjectTypeName := 'MyProduct';
							MpPickRegCreatePlaceholder.Parameters.Translation.X := tablicaPlace[1];
							MpPickRegCreatePlaceholder.Parameters.Translation.Y := PlaceY; // in the middle of conveyor width
							MpPickRegCreatePlaceholder.Create := TRUE;
							iteracja := 2;
							abc := 0;
						2:
							MpPickRegCreatePlaceholder.Parameters.LatchedConveyor.Position := PlaceConveyorPosition;
							MpPickRegCreatePlaceholder.Parameters.Mode := mpPICK_CREATE_SINGLEITEM_PLACEH;
							MpPickRegCreatePlaceholder.Parameters.ObjectTypeName := 'MyProduct';
							MpPickRegCreatePlaceholder.Parameters.Translation.X := tablicaPlace[2];
							MpPickRegCreatePlaceholder.Parameters.Translation.Y := PlaceY; // in the middle of conveyor width
							MpPickRegCreatePlaceholder.Create := TRUE;
							iteracja := 3;
							abc := 0;

						3:
							MpPickRegCreatePlaceholder.Parameters.LatchedConveyor.Position := PlaceConveyorPosition;
							MpPickRegCreatePlaceholder.Parameters.Mode := mpPICK_CREATE_SINGLEITEM_PLACEH;
							MpPickRegCreatePlaceholder.Parameters.ObjectTypeName := 'MyProduct';
							MpPickRegCreatePlaceholder.Parameters.Translation.X := tablicaPlace[3];
							MpPickRegCreatePlaceholder.Parameters.Translation.Y := PlaceY; // in the middle of conveyor width
							MpPickRegCreatePlaceholder.Create := TRUE;
							iteracja := 4;
							abc := 0;
						4:
							abc :=0;
					END_CASE;
				ELSE
					MpPickRegCreatePlaceholder.Create := FALSE;

					abc :=1;
				END_IF

//
//		//	ELSE
//
//			END_IF

//			MpPickRegGetObjectsContainer.Parameters.DataAddress := ADR(gContainerInfo);
//			MpPickRegGetObjectsContainer.Parameters.GetMode := mpPICK_GET_CONTAINER_CONTENT;
//			MpPickRegGetObjectsContainer.Parameters.ObjectPositionId := ContainerID;
//			MpPickRegGetObjectsContainer.Parameters.ObjectTypeName := 'MyContainer';
//			MpPickRegGetObjectsContainer.Parameters.NumberOfObjectPositions := 4;
//			MpPickRegGetObjectsContainer.MpLink := ADR(gPlaceRegister);
//			MpPickRegGetObjectsContainer();

//			// Konfiguracja bloku GetObjects1
//			GetObjects1.Parameters.DataAddress :=ADR(g
//			GetObjects1.Parameters.GetMode := mpPICK_GET_ALL_SINGLEITEMS;
//			GetObjects1.Parameters.ObjectTypeName := WSTRING_TO_STRING("MyProduct");
//			GetObjects1.Parameters.ObjectPositionId := LREAL_TO_UDINT(MpPickRegCreatePlaceholder.Parameters.LatchedConveyor.Position);
//
//			// Aktywacja bloku
//			GetObjects1.Enable := TRUE;
//
//			// Czekanie na zakoñczenie operacji
//			IF GetObjects1.CommandDone THEN
//				ilosc1 := GetObjects1.ObjectPositionsFound; // Pobieranie liczby znalezionych obiektów
//				GetObjects1.Enable := FALSE;  // Zatrzymanie bloku po zakoñczeniu operacji
//			END_IF;

		P_ERROR:
			Error := TRUE;
			ReadyPlaceReg := FALSE;

	END_CASE;

	(* FB calls *)
	MpPickRegister_0.MpLink := ADR(gPlaceRegister);
	MpPickRegister_0();

	MpPickRegCreatePlaceholder.MpLink := ADR(gPlaceRegister);
	MpPickRegCreatePlaceholder();

	GetObjects1.MpLink := ADR(gPlaceRegister);
	GetObjects1;

END_PROGRAM
```

### Program Logical/PickAndPlace/Program (IEC)

#### Types.typ
```iecst
TYPE
	Krok :
		(
		HOME,
		POWER,
		PROG,
		CHECK,
		RUCH
		);
END_TYPE
```

#### Variables.var
```iecst
VAR
	AxisParam1 : MpAxisBasicParType;
	AxisParam2 : MpAxisBasicParType;
	AxisParam3 : MpAxisBasicParType;
	AxisParam4 : MpAxisBasicParType;
	FB_Axis1 : MpAxisBasic;
	FB_Axis2 : MpAxisBasic;
	FB_Axis3 : MpAxisBasic;
	FB_Axis4 : MpAxisBasic;
	KrokXYZ : Krok;
END_VAR
```

#### Main.st
```iecst
PROGRAM _INIT
	KrokXYZ := CHECK;

	FB_Axis1.Enable := TRUE;
	FB_Axis2.Enable := TRUE;
	FB_Axis3.Enable := TRUE;

END_PROGRAM

PROGRAM _CYCLIC
//	CASE KrokXYZ OF
//		CHECK:
//			IF 	manXYZ THEN
//				FB_Axis1.Home := FALSE;
//				FB_Axis2.Home := FALSE;
//				FB_Axis3.Home := FALSE;
//
//				FB_Axis1.Power := FALSE;
//				FB_Axis2.Power := FALSE;
//				FB_Axis3.Power := FALSE;
//
//				FB_Axis1.Enable := FALSE;
//				FB_Axis2.Enable := FALSE;
//				FB_Axis3.Enable := FALSE;
//
//				KrokXYZ := WAIT;
//			END_IF;
//			FB_Axis1.MoveAbsolute :=FALSE;
//			FB_Axis2.MoveAbsolute :=FALSE;
//			FB_Axis3.MoveAbsolute :=FALSE;
//			IF FB_Axis1.Active AND FB_Axis2.Active AND FB_Axis3.Active THEN
//				KrokXYZ := POWER;
//			END_IF;
//		POWER:
//			FB_Axis1.Power := TRUE;
//			FB_Axis2.Power := TRUE;
//			FB_Axis3.Power := TRUE;
//
//			IF FB_Axis1.PowerOn AND FB_Axis2.PowerOn AND FB_Axis3.PowerOn THEN
//				KrokXYZ := HOME;
//			END_IF;
		(*HOME:*)
	AxisParam1.Homing.Mode := mcHOMING_ABSOLUTE;
	AxisParam1.Homing.Position := -472776.56;
	AxisParam2.Homing.Mode := mcHOMING_ABSOLUTE;
	AxisParam2.Homing.Position := 77660.78;
	AxisParam3.Homing.Mode := mcHOMING_ABSOLUTE;
	AxisParam3.Homing.Position := 3712.2;

//			IF FB_Axis1.IsHomed AND FB_Axis2.IsHomed AND FB_Axis3.IsHomed THEN
//				FB_Axis1.Home := FALSE;
//				FB_Axis2.Home := FALSE;
//				FB_Axis3.Home := FALSE;
//
//				setAxis1:=  FB_Axis1.Position;
//				setAxis2 := FB_Axis2.Position;
//				setAxis3 := FB_Axis3.Position;
//				KrokXYZ := PROG;
//
//			END_IF;
//		PROG:
//			(*DeltaParameters.ProgramName := 'Robotic.st';*)
//			IF 	manXYZ THEN
//				KrokXYZ := CHECK;
//			END_IF;
//			AxisParam1.Position := setAxis1;
//			AxisParam2.Position := setAxis2;
//			AxisParam3.Position := setAxis3;
//			IF saveChanges THEN
//				KrokXYZ:=RUCH;
//			END_IF;
//		RUCH:
//			IF  FB_Axis1.Position<> setAxis1 THEN
//				FB_Axis1.MoveAbsolute := TRUE;
//			END_IF;
//			IF FB_Axis2.Position <> setAxis2 THEN
//				FB_Axis2.MoveAbsolute := TRUE;
//			END_IF;
//			IF FB_Axis3.Position <> setAxis3 THEN
//				FB_Axis3.MoveAbsolute := TRUE;
//			END_IF;
//			saveChanges :=FALSE;
//
//			KrokXYZ:=FLAGI;
//		FLAGI:
//			IF FB_Axis1.Position = setAxis1 AND FB_Axis2.Position = setAxis2 AND FB_Axis3.Position = setAxis3 THEN
//				KrokXYZ:=CHECK;
//			END_IF
//		WAIT:
//			IF NOT manXYZ THEN
//				FB_Axis1.Enable := TRUE;
//				FB_Axis2.Enable := TRUE;
//				FB_Axis3.Enable := TRUE;
//				FB_Axis4.Enable := TRUE;
//				KrokXYZ:= CHECK;
//			END_IF
//	END_CASE;

	FB_Axis1.MpLink     := ADR(gAxisQ1);
	FB_Axis1.Parameters := ADR(AxisParam1);
	FB_Axis1();

	FB_Axis2.MpLink     := ADR(gAxisQ2);
	FB_Axis2.Parameters := ADR(AxisParam2);
	FB_Axis2();

	FB_Axis3.MpLink     := ADR(gAxisQ3);
	FB_Axis3.Parameters := ADR(AxisParam3);
	FB_Axis3();

	FB_Axis4.MpLink     := ADR(gAxisQ4);
	FB_Axis4.Parameters := ADR(AxisParam4);
	FB_Axis4();
//

END_PROGRAM

PROGRAM _EXIT
	(* Insert code here *)

END_PROGRAM
```

### Program Logical/PickAndPlace/TCPXYZ

#### Types.typ
```iecst
TYPE
	Krok :
		(
		HOME,
		POWER,
		PROG,
		CHECK,
		RUCH,
		FLAGI,
		WAIT,
		POWERAXIS,
		HOMEAXIS,
		CHECKAXIS,
		CHECKDELTA,
		ENABLE,
		ON,
		HOMEFLAG,
		OFF,
		MODE,
		PRGMECH,
		AUTOMODE
	);
END_TYPE
```

#### Variables.var
```iecst
VAR
	MpDelta4Axis_0 : MpDelta4Axis;
	MpAxisBasic_1 : MpAxisBasic;
	MpAxisBasic_0 : MpAxisBasic;
	KrokXYZ : Krok;
	KrokConv : Krok;
	HomePosition : BOOL;
	HomeButton : BOOL;
	FB_Axis4 : MpAxisBasic;
	FB_Axis3 : MpAxisBasic;
	FB_Axis2 : MpAxisBasic;
	FB_Axis1 : MpAxisBasic;
	DeltaParameters : MpDelta4AxisParType;
	ConveyerButton : BOOL := FALSE;
	AxisParameters_1 : MpAxisBasicParType;
	AxisParameters_0 : MpAxisBasicParType;
	AxisParam4 : MpAxisBasicParType;
	AxisParam3 : MpAxisBasicParType;
	AxisParam2 : MpAxisBasicParType;
	AxisParam1 : MpAxisBasicParType;
	FB_AlarmHistory : MpAlarmXHistory;
	FB_AlarmCore : MpAlarmXCore;
END_VAR
```

#### Main.st
```iecst
PROGRAM _INIT
	MpDelta4Axis_0.Override := 100.0;
	//	MpDelta4Axis_0.Enable := TRUE;
	AxisParameters_0.Velocity     := 5.0;
	AxisParameters_0.Acceleration := 50.0;
	AxisParameters_0.Deceleration := 50.0;
	FB_AlarmCore.MpLink := ADR(gAlarmXCore);
	FB_AlarmCore.Enable := TRUE;
	FB_AlarmHistory.MpLink := ADR(gAlarmXHistory);
	FB_AlarmHistory.Enable := TRUE;

	AxisParameters_1.Velocity     := 130.0;
	AxisParameters_1.Acceleration := 50.0;
	AxisParameters_1.Deceleration := 50.0;

//	AxisParam1.Homing.Mode := mcHOMING_ABSOLUTE;
//	AxisParam1.Homing.Position := -472771;
//	AxisParam2.Homing.Mode := mcHOMING_ABSOLUTE;
//	AxisParam2.Homing.Position := 77669;
//	AxisParam3.Homing.Mode := mcHOMING_ABSOLUTE;
//	AxisParam3.Homing.Position := 3718;

	KrokConv:= ENABLE;
	KrokXYZ := ENABLE;
	gAxisQ1;
	gAxisQ2;
	gAxisQ3;
	gAxisQ4;
END_PROGRAM

PROGRAM _CYCLIC
//	CASE KrokConv OF
//		ENABLE:
//			MpAxisBasic_0.Enable :=TRUE;
//			MpAxisBasic_1.Enable :=TRUE;
//			KrokConv:= CHECK;
//		CHECK:
//			IF MpAxisBasic_0.Active AND MpAxisBasic_1.Active THEN
//				MpAxisBasic_0.Power :=TRUE;
//				MpAxisBasic_1.Power :=TRUE;
//				KrokConv := POWER;
//			END_IF
//		POWER:
//			IF MpAxisBasic_0.PowerOn THEN
//				MpAxisBasic_0.Home := TRUE;
//				KrokConv := PROG;
//			END_IF
//		PROG:
//			IF MpAxisBasic_0.IsHomed THEN
//				IF ConveyerButton THEN
//					MpAxisBasic_0.MoveVelocity := TRUE;
//					KrokConv:= FLAGI;
//				ELSE
//					MpAxisBasic_0.MoveVelocity :=FALSE;
//				END_IF;
//
//			END_IF
//		FLAGI:
//			IF NOT ConveyerButton OR NOT Mode THEN
//				MpAxisBasic_0.MoveVelocity :=FALSE;
//				MpAxisBasic_0.Home:=FALSE;
//				MpAxisBasic_0.Power:=FALSE;
//				MpAxisBasic_0.Enable:=FALSE;
//				KrokConv:= ON;
//			END_IF;
//	END_CASE

	CASE KrokXYZ OF
		ENABLE:
			FB_Axis1.Enable :=TRUE;
			FB_Axis2.Enable :=TRUE;
			FB_Axis3.Enable :=TRUE;
			FB_Axis4.Enable :=TRUE;
			MpAxisBasic_0.Enable:=TRUE;
			MpAxisBasic_1.Enable:=TRUE;

			KrokXYZ := POWERAXIS;

		POWERAXIS:
			IF FB_Axis1.Active AND FB_Axis2.Active AND FB_Axis3.Active THEN
				FB_Axis1.Power := TRUE;
				FB_Axis2.Power := TRUE;
				FB_Axis3.Power := TRUE;
				FB_Axis4.Power := TRUE;
				MpAxisBasic_0.Power := TRUE;
				MpAxisBasic_1.Power:=TRUE;
				KrokXYZ := HOMEAXIS;
			END_IF

		HOMEAXIS:
			IF FB_Axis1.PowerOn AND FB_Axis2.PowerOn AND FB_Axis3.PowerOn THEN
				FB_Axis1.Home := TRUE;
				FB_Axis2.Home := TRUE;
				FB_Axis3.Home := TRUE;
				FB_Axis4.Home := TRUE;
				MpAxisBasic_0.Home := TRUE;
				MpAxisBasic_1.Home:=TRUE;

				KrokXYZ := CHECKAXIS;
			END_IF

		CHECKAXIS:
			IF FB_Axis1.IsHomed AND FB_Axis2.IsHomed AND FB_Axis3.IsHomed THEN
				FB_Axis1.Home := FALSE;
				FB_Axis2.Home := FALSE;
				FB_Axis3.Home := FALSE;
				FB_Axis4.Home := FALSE;
				MpAxisBasic_0.Home:= FALSE;
				MpAxisBasic_1.Home:=FALSE;
				FB_Axis1.Enable :=FALSE;
				FB_Axis2.Enable :=FALSE;
				FB_Axis3.Enable :=FALSE;
				FB_Axis4.Enable :=FALSE;

				KrokXYZ := CHECKDELTA;
			END_IF

		CHECKDELTA:
			IF NOT FB_Axis1.Active AND NOT FB_Axis2.Active AND NOT FB_Axis3.Active THEN
				MpDelta4Axis_0.Enable := TRUE;
				KrokXYZ := CHECK;
			END_IF
		CHECK:
			MpDelta4Axis_0.MoveDirect := FALSE;
			MpDelta4Axis_0.MoveLinear := FALSE;
			IF MpDelta4Axis_0.Active AND MpDelta4Axis_0.IsHomed AND MpDelta4Axis_0.PowerOn THEN
				KrokXYZ := HOME;
			END_IF;

			IF MpDelta4Axis_0.Active THEN
				KrokXYZ := POWER;
			END_IF;
		POWER:
			MpDelta4Axis_0.Power := TRUE;
			IF MpDelta4Axis_0.PowerOn THEN
				KrokXYZ := HOME;
			END_IF;
		HOME:
			IF MpDelta4Axis_0.IsHomed THEN
				setX := MpDelta4Axis_0.X;
				setY :=  MpDelta4Axis_0.Y;
				setZ := MpDelta4Axis_0.Z;

				setAxis1 := MpDelta4Axis_0.Info.JointAxisPosition[0];
				setAxis2 := MpDelta4Axis_0.Info.JointAxisPosition[1];
				setAxis3 := MpDelta4Axis_0.Info.JointAxisPosition[2];

				KrokXYZ := PROG;
			END_IF;
		PROG:
			IF Mode AND ConveyerButton THEN
				MpAxisBasic_0.MoveVelocity := TRUE;
			ELSIF NOT Mode OR NOT ConveyerButton THEN
				MpAxisBasic_0.MoveVelocity :=FALSE;
			END_IF;
			IF NOT Mode THEN
				MpDelta4Axis_0.MoveDirect := FALSE;
				MpDelta4Axis_0.MoveLinear := FALSE;
				IF MpAxisBasic_0.IsHomed THEN
					MpAxisBasic_0.Home:= FALSE;
					ReadyMechanics := TRUE;
					KrokXYZ := PRGMECH;
				END_IF;
			END_IF
			IF ABS(MpDelta4Axis_0.Info.JointAxisPosition[0])<0.01 AND ABS(MpDelta4Axis_0.Info.JointAxisPosition[1])<0.01 AND ABS(MpDelta4Axis_0.Info.JointAxisPosition[2])<0.01 THEN
				HomePosition :=TRUE;
			ELSE
				HomePosition :=FALSE;
			END_IF

			IF TCP = TRUE AND HomeButton = FALSE THEN
				DeltaParameters.CoordSystem := 1;
				DeltaParameters.Position[0] := setX;
				DeltaParameters.Position[1]:= setY;
				DeltaParameters.Position[2]:= setZ;
				DeltaParameters.Position[3]:= 0;

			ELSIF TCP = FALSE AND HomeButton =FALSE THEN
				DeltaParameters.CoordSystem := 0;
				DeltaParameters.Position[0] := setAxis1;
				DeltaParameters.Position[1]:= setAxis2;
				DeltaParameters.Position[2]:= setAxis3;
				DeltaParameters.Position[3]:= 0;

			ELSIF HomeButton THEN
				KrokXYZ :=HOMEFLAG;
			END_IF;

			IF saveChanges THEN
				KrokXYZ:=RUCH;
			END_IF;

		RUCH:

			IF DeltaParameters.CoordSystem = 1 THEN
				MpDelta4Axis_0.MoveLinear := TRUE;
			ELSE
				MpDelta4Axis_0.MoveDirect := TRUE;
			END_IF;

			saveChanges :=FALSE;
			KrokXYZ:=FLAGI;
		FLAGI:
			IF ABS(MpDelta4Axis_0.Info.JointAxisPosition[0])<0.01 AND ABS(MpDelta4Axis_0.Info.JointAxisPosition[1])<0.01 AND ABS(MpDelta4Axis_0.Info.JointAxisPosition[2])<0.01 THEN
				HomePosition := TRUE;
			ELSE
				HomePosition := FALSE;
			END_IF
			IF DeltaParameters.CoordSystem = 0 AND ABS(MpDelta4Axis_0.Info.JointAxisPosition[0]-setAxis1)<0.01 AND ABS(MpDelta4Axis_0.Info.JointAxisPosition[1]-setAxis2)<0.01 AND ABS(MpDelta4Axis_0.Info.JointAxisPosition[2]-setAxis3)<0.01 THEN
				KrokXYZ:=CHECK;
			END_IF

			IF DeltaParameters.CoordSystem = 1 AND ABS(MpDelta4Axis_0.X-setX)<0.01 AND ABS(MpDelta4Axis_0.Y - setY)<0.01 AND ABS(MpDelta4Axis_0.Z-setZ)<0.01 THEN
				KrokXYZ:=CHECK;
			END_IF
		HOMEFLAG:
			DeltaParameters.CoordSystem := 0;
			DeltaParameters.Position[0] := 0;
			DeltaParameters.Position[1]:= 0;
			DeltaParameters.Position[2]:= 0;
			DeltaParameters.Position[3]:= 0;
			MpDelta4Axis_0.MoveDirect := TRUE;
			IF DeltaParameters.CoordSystem = 0 AND ABS(MpDelta4Axis_0.Info.JointAxisPosition[0])<0.01 AND ABS(MpDelta4Axis_0.Info.JointAxisPosition[1])<0.01 AND ABS(MpDelta4Axis_0.Info.JointAxisPosition[2])<0.01 THEN
				HomeButton:=FALSE;
				KrokXYZ:=CHECK;
			END_IF
		PRGMECH:

			MpAxisBasic_0.MoveVelocity := TRUE;
			IF CmdStart AND ReadyToStart THEN
				KrokXYZ:= AUTOMODE;
			END_IF
			IF Mode THEN
				MpAxisBasic_0.MoveVelocity :=FALSE;
				ReadyMechanics :=FALSE;
				KrokXYZ :=	PROG;
			END_IF
		AUTOMODE:
			IF Mode THEN
				MpAxisBasic_0.MoveVelocity :=FALSE;
				ReadyMechanics :=FALSE;
				KrokXYZ :=	PROG;
			END_IF
	END_CASE;

	ReadyToStart := ReadyMechanics AND ReadyPickReg AND ReadyPlaceReg AND ReadyPickCore;

	FB_AlarmCore();
	FB_AlarmHistory();

	IF MpDelta4Axis_0.Error THEN
		MpAlarmXSet(gAlarmXCore,'DeltaError');
	ELSE
		MpAlarmXReset(gAlarmXCore,'DeltaError');
	END_IF;

	IF MpAxisBasic_0.Error THEN
		MpAlarmXSet(gAlarmXCore,'ConveyorAxisError');
	ELSE
		MpAlarmXReset(gAlarmXCore,'ConveyorAxisError');
	END_IF;

	IF FB_Axis1.Error THEN
		MpAlarmXSet(gAlarmXCore,'DeltaAxis1Error');
	ELSE
		MpAlarmXReset(gAlarmXCore,'DeltaAxis1Error');
	END_IF;

	IF FB_Axis2.Error THEN
		MpAlarmXSet(gAlarmXCore,'DeltaAxis2Error');
	ELSE
		MpAlarmXReset(gAlarmXCore,'DeltaAxis2Error');
	END_IF;

	IF FB_Axis3.Error THEN
		MpAlarmXSet(gAlarmXCore,'DeltaAxis3Error');
	ELSE
		MpAlarmXReset(gAlarmXCore,'DeltaAxis3Error');
	END_IF;

	IF FB_Axis4.Error THEN
		MpAlarmXSet(gAlarmXCore,'DeltaVirtualAxisError');
	ELSE
		MpAlarmXReset(gAlarmXCore,'DeltaVirtualAxisError');
	END_IF;

	FB_Axis1.MpLink     := ADR(gAxisQ1);
	FB_Axis1.Parameters := ADR(AxisParam1);
	FB_Axis1();

	FB_Axis2.MpLink     := ADR(gAxisQ2);
	FB_Axis2.Parameters := ADR(AxisParam2);
	FB_Axis2();

	FB_Axis3.MpLink     := ADR(gAxisQ3);
	FB_Axis3.Parameters := ADR(AxisParam3);
	FB_Axis3();

	FB_Axis4.MpLink     := ADR(gAxisQ4);
	FB_Axis4.Parameters := ADR(AxisParam4);
	FB_Axis4();

	MpAxisBasic_0.MpLink     := ADR(gAxis_1);
	MpAxisBasic_0.Parameters := ADR(AxisParameters_0);
	MpAxisBasic_0();

	MpAxisBasic_1.MpLink     := ADR(gAxis_2);
	MpAxisBasic_1.Parameters := ADR(AxisParameters_1);
	MpAxisBasic_1();

	MpDelta4Axis_0.Parameters := ADR(DeltaParameters);
	MpDelta4Axis_0.MpLink := ADR(g4AxDeltaA);
	MpDelta4Axis_0();

	PickConveyorPosition  := MpAxisBasic_0.Position;
	PlaceConveyorPosition := MpAxisBasic_1.Position;
END_PROGRAM

//PROGRAM _EXIT
//	MpDelta4Axis_0.Enable := FALSE;
//	MpDelta4Axis_0.MpLink := 0;
//END_PROGRAM
```

- Visualisation Logical/mappView (not shown)

### Robotics.st
```iecst
VAR CONSTANT
P1 : McPointType := (Pos:=(X:=140.4, Y:=0, Z:=97));
P2 : McPointType := (Pos:=(X:=-83, Y:=-195, Z:=80));
P3 : McPointType := (Pos:=(X:=-83, Y:=-195, Z:=42));
P5 : McPointType := (Pos:=(X:=-83, Y:=-30, Z:=80));
P6 : McPointType := (Pos:=(X:=-83, Y:=-30, Z:=39));
P8 : McPointType := (Pos:=(X:=-45, Y:=-195, Z:=80));
P9 : McPointType := (Pos:=(X:=-45, Y:=-195, Z:=47));
	Gripper := FALSE;
	END_VAR

	PROGRAM _MAIN
	Feedrate(5000);   //move with reduced speeda
	MoveJ(P1);        //move system to point P1
	MoveJ(P2);        //move system to point P2
	MoveJ(P3);
	Gripper := TRUE;
	MoveJ(P2);
	MoveJ(P5);
	MoveJ(P6);
	Gripper := FALSE;
	MoveJ(P5);
	MoveJ(P8);
	MoveJ(P9);
	Gripper := TRUE;
	MoveJ(P8);
	MoveJ(P5);
	MoveJ(P6);
	Gripper := FALSE;
	MoveJ(P5);
	WaitTime(3);        //wait for 3 seconds
	MoveJ(P1);        //move back to origin position
	END_PROGRAM
```

### Program Logical/Program

#### Types.typ
```iecst
TYPE
	DeltaState :
		(
		Delta_Idle,
		Delta_Power,
		Delta_Home,
		Delta_Ready,
		Delta_Error,
		Delta_Move
	);
END_TYPE
```

#### Main.st
```iecst
PROGRAM _INIT

(*
	MpDelta3Axis_0.Enable := TRUE;
	MpDelta3Axis_0.Override := 100.0;
	DeltaParameters.ProgramName := 'Robotic.st';    //File stored on FileDevice

	FB_Axis_1.Enable := TRUE;
	FB_Axis_2.Enable := TRUE;
	FB_Axis_3.Enable := TRUE;

	AxisParam_1.Velocity := 10;
	AxisParam_1.Distance := 50;
	AxisParam_1.Position := 100;*)
END_PROGRAM

PROGRAM _CYCLIC
		(*
    MpDelta3Axis_0.Parameters := ADR(DeltaParameters);

	FB_Axis_1.MpLink := ADR(gAxisQ1);
	FB_Axis_2.MpLink := ADR(gAxisQ2);
	FB_Axis_3.MpLink := ADR(gAxisQ3);

	FB_Axis_1.Parameters := ADR(AxisParam_1);
	FB_Axis_2.Parameters := ADR(AxisParam_1);
	FB_Axis_3.Parameters := ADR(AxisParam_1);

	FB_Axis_1();
	FB_Axis_2();
	FB_Axis_3();

	MpDelta3Axis_0();
	//VisuPos[0] := LREAL_TO_REAL(MpDelta3Axis_0.Info.JointAxisPosition[0]);
	VisuPos[0] := LREAL_TO_REAL(MpDelta3Axis_0.Info.JointAxisPosition[0]);
	VisuPos[1] := LREAL_TO_REAL(MpDelta3Axis_0.Info.JointAxisPosition[1]);
	VisuPos[2] := LREAL_TO_REAL(MpDelta3Axis_0.Info.JointAxisPosition[2]);

	VisuPos[0] := LREAL_TO_REAL(FB_Axis_1.Position);
	VisuPos[1] := LREAL_TO_REAL(FB_Axis_2.Position);
	VisuPos[2] := LREAL_TO_REAL(FB_Axis_3.Position);

	IF MpDelta3Axis_0.Error THEN
		DeltaStep := Delta_Error;
	END_IF;

	CASE DeltaStep OF
		Delta_Idle://IDLE state - all comands reset
			MpDelta3Axis_0.Power := FALSE;
			MpDelta3Axis_0.Home := FALSE;
			MpDelta3Axis_0.MoveProgram := FALSE;

			IF diDeltaOn AND	MpDelta3Axis_0.Info.ReadyToPowerOn  THEN
				DeltaStep := Delta_Power;
			END_IF;
		Delta_Power://Power state - comand power is active - waiting for PowerON flag
			 MpDelta3Axis_0.Power := TRUE;
			IF MpDelta3Axis_0.PowerOn THEN
				DeltaStep := Delta_Home;
			END_IF;
		Delta_Home://Homae state- comand gome is active - waiting for is Homed flag
			 MpDelta3Axis_0.Home:= TRUE;
			IF MpDelta3Axis_0.IsHomed THEN
				DeltaStep := Delta_Ready;
			END_IF;
		Delta_Ready://Ready state
			MpDelta3Axis_0.Home := FALSE;
			MpDelta3Axis_0.MoveProgram := FALSE;

			IF   NOT diDeltaOn	THEN
				DeltaStep := Delta_Idle;
			END_IF;
		Delta_Error://Error state - all caomends reset - waiting for Error flag to be reset
			MpDelta3Axis_0.Power := FALSE;
			MpDelta3Axis_0.Home := FALSE;
			MpDelta3Axis_0.MoveProgram := FALSE;

			IF NOT MpDelta3Axis_0.Error THEN
				DeltaStep := Delta_Idle;
			END_IF;

	END_CASE;
     	 	*)
END_PROGRAM

PROGRAM _EXIT
	(* Insert code here *)

END_PROGRAM
```

Listed in the project but not available here: Logical/Global.typ, Logical/PickAndPlace/UserLibraries, Logical/PickAndPlace/Scene
